	    // decoding of EFPC modus
	    CASE BYTE_TO_INT(#FML_REF.FPCS_Modus) OF
	        0: (* old style *)
	            (* 
	            -------------- Byte 1 --------------- Byte 2 ---------------------- Byte 3/4 ------------------- Byte 5..8 ----
	            |  8  7  6  5  4  |  3  2  1  0  |              | 15 14 13 12 |  11  | 10 9 8 7 6 5 4 3 2 1 0 |               |
	            |    FPCS Modus   |     res      |   Subindex   |      AK     |  SPM |        PNU             |     Value     |
	            ---------------------------------------------------------------------------------------------------------------     
	            AK:  Response Identifier (Antwortkennung)
	            SPM: NOT used
	            PNU: Parameternummer / Parameter-Number 
	            *)
	            // Byte1
	            // zero in this CASE
	            // Byte2  
	            #FML_REF.ActSubindex := #FML_REF.InData.FPC[2];
	            
	            // Byte3/4
	            #BByte2[1] := #FML_REF.InData.FPC[3];
	            #BByte2[2] := #FML_REF.InData.FPC[4];
	            #Resp_Identifier := WORD_TO_INT(SHR(IN := (#_Word AND 2#1111000000000000), N := 12));
	            #FML_REF.ActPNU := #_Word AND 2#0000011111111111;
	            
	            // Byte 5..8 parameter value
	            #BByte4[1] := #FML_REF.InData.FPC[5];
	            #BByte4[2] := #FML_REF.InData.FPC[6];
	            #BByte4[3] := #FML_REF.InData.FPC[7];
	            #BByte4[4] := #FML_REF.InData.FPC[8];
	            #FML_REF.ParamValueRD := #_DINT;
	            
	        1, 2, 3:(* modus: 1 = PNU extended; 2 = KO; 3 = CAN Objects *)
	            (* 
	            -------------- Byte 1 --------------- Byte 2 ------------------- Byte 3/4----------------- Byte 5..8 ----
	            |   7  6  5  4  |  3  2  1  0  |              | 15 14 13 12 11 10 9 8 7 6 5 4 3 2 1 0 |               |
	            |  FPCS Modus   |     AK       |   Subindex   |   PNU extended or KO or CAN Object    |     Value     |
	            -------------------------------------------------------------------------------------------------------       
	            AK:  Response Identifier (Antwortkennung)
	            *)
	            
	            // Byte 1 FPCS
	            #Resp_Identifier := WORD_TO_INT(#FML_REF.InData.FPC[1] AND 2#00001111);
	            
	            // Byte 2 Subindex
	            #FML_REF.ActSubindex := #FML_REF.InData.FPC[2];
	            
	            // Byte 3+4 **PKE/ PNU/ KO/ CAN**
	            #BByte2[1] := #FML_REF.InData.FPC[3];
	            #BByte2[2] := #FML_REF.InData.FPC[4];
	            #FML_REF.ActPNU := #_Word;
	            
	            // Byte 5..8 parameter value
	            #BByte4[1] := #FML_REF.InData.FPC[5];
	            #BByte4[2] := #FML_REF.InData.FPC[6];
	            #BByte4[3] := #FML_REF.InData.FPC[7];
	            #BByte4[4] := #FML_REF.InData.FPC[8];
	            #FML_REF.ParamValueRD := #_DINT;
	            
	        4, 5:(* FPCS_Modus 4=Parameter File; 5=Firmware File *)
	            (*
	            ------ BYTE 1 ------------|-- BYTE 2 -|--BYTE 3..8 ---|
	            | 7  6  5  4 | 3  2  1  0 |           |               |
	            | FPCS Modus |   res      | Packet-ID |  6 BYTE Data  |
	            -------------------------------------------------------        
	              Packet-ID: -------------- BYTE 2 ----------
	                         | 7    6    5  | 4  3  2  1  0 |
	                         | Control Bits |   Sequence-Nr |
	                         -------------------------------- 
	            *)
	            // Byte 1 FPCS
	            #Resp_Identifier := WORD_TO_INT(#FML_REF.InData.FPC[1] AND 2#00001111);
	            #FML_REF.RespID := #Resp_Identifier;
	            
	            //---- Byte 2 Packet-ID ----    
	            #FML_REF.FPCS_Packet.BitSequenceNr := WORD_TO_INT(#FML_REF.InData.FPC[2] AND 2#00011111);
	            #FML_REF.FPCS_Packet.Control := WORD_TO_INT(SHR(IN := (#FML_REF.InData.FPC[2] AND 2#11100000), N := 5));
	            //---- Byte 3..8 Data ----
	            #FML_REF.FPCS_Packet.Data[1] := #FML_REF.InData.FPC[3];
	            #FML_REF.FPCS_Packet.Data[2] := #FML_REF.InData.FPC[4];
	            #FML_REF.FPCS_Packet.Data[3] := #FML_REF.InData.FPC[5];
	            #FML_REF.FPCS_Packet.Data[4] := #FML_REF.InData.FPC[6];
	            #FML_REF.FPCS_Packet.Data[5] := #FML_REF.InData.FPC[7];
	            #FML_REF.FPCS_Packet.Data[6] := #FML_REF.InData.FPC[8];
	            
	            
	        ELSE (* not implemented *)
	            #FPC_MAPPING := FALSE; (* Execution was not correct *)
	            RETURN;
	    END_CASE;
	    
	    CASE #Resp_Identifier OF
	        0, 3:(* No Transmission or Active*)
	            #FML_REF.Done := FALSE;
	            #FML_REF.Err := FALSE;
	            #FML_REF.ActPNU := 0;
	            #FML_REF.ActSubindex := 0;
	            #FML_REF.ParamValueRD := 0;
	            #FML_REF.DatatypeRD := 0;
	            
	            
	        1, 4:(* Word Parameter transmittead*)
	            #FML_REF.Done := TRUE;
	            #FML_REF.Err := FALSE;
	            #FML_REF.ParamValueRD := #_DINT;
	            #FML_REF.DatatypeRD := 2;
	            
	        2, 5: (*DWord Parameter transmitted*)
	            #FML_REF.Done := true;
	            #FML_REF.Err := FALSE;
	            #FML_REF.ParamValueRD := #_DINT;
	            #FML_REF.DatatypeRD := 4;
	            
	        7:(* Transmission Failed*)
	            #FML_REF.Done := TRUE;
	            #FML_REF.Err := TRUE;
	            #FML_REF.DatatypeRD := 0;
	            #FML_REF.ParamValueRD := 0;
	            #FML_REF.ActPNU := 0;
	            
	            
	        11, 12: (*BYTE Parameter transmitted*)
	            #FML_REF.Done := TRUE;
	            #FML_REF.Err := False;
	            #FML_REF.DatatypeRD := 1;
	            #FML_REF.ParamValueRD := #_DINT;
	            
	        ELSE (* not specified*)
	            #FML_REF.Done := false;
	            #FML_REF.Err := TRUE;
	            #FML_REF.ParamValueRD := 0;
	    END_CASE;
	    
	    #FPC_MAPPING := TRUE; (* Execution was correct *)
	    RETURN;
	    
	(* MAP OUTPUTS *)
	ELSE
	    
	    IF #FML_REF.DeviceType = 'SFC_DC' OR #FML_REF.DeviceType = 'MTR_DCI' THEN
	        IF #FML_REF.ReqID = 8 THEN // write
	            IF BYTE_TO_INT(#FML_REF.Subindex) > 0 THEN
	                CASE BYTE_TO_INT(#FML_REF.DatatypeWR) OF
	                    1:
	                        #FML_REF.ReqID := 12;     //Array-Byte
	                    2:
	                        #FML_REF.ReqID := 7;      //Array-Wort
	                    4:
	                        #FML_REF.ReqID := 8;      //Array-Doppelwort
	                    ELSE
	                        #FPC_MAPPING := FALSE; (* wrong data type*)
	                        RETURN;
	                END_CASE;
	            END_IF;
	            (*WRITE SINGLE PARAMETER*)
	            IF #FML_REF.Subindex = 0 THEN
	                CASE BYTE_TO_INT(#FML_REF.DatatypeWR) OF
	                    1:
	                        #FML_REF.ReqID := 11;       // Single-Byte
	                    2:
	                        #FML_REF.ReqID := 2;        // Single-Wort
	                    4:
	                        #FML_REF.ReqID := 3;        // Single-Doppelwort
	                    ELSE
	                        #FPC_MAPPING := FALSE; (* wrong data type*)
	                        RETURN;
	                END_CASE;
	            END_IF;
	            
	        ELSIF #FML_REF.ReqID = 6 THEN
	            (* READ ARRAY PARAMETER *)
	            IF BYTE_TO_INT(#FML_REF.Subindex) > 0 THEN
	                #FML_REF.ReqID := 6;
	            END_IF;
	            (* READ SINGLE PARAMETER *)
	            IF #FML_REF.Subindex = 0 THEN
	                #FML_REF.ReqID := 1;
	            END_IF;
	        ELSE
	            ;// not specified
	        END_IF;
	    END_IF;
	    (* create request identifier *)
	    #Req_Identifier := #FML_REF.ReqID;
	    
	    CASE BYTE_TO_INT(#FML_REF.FPCC_Modus) OF
	        0: (* old style *)
	            (* 
	            -------------- Byte 1 --------------- Byte 2 ---------------------- Byte 3 --------------------- Byte 5..8 ----
	            |  8  7  6  5  4  |  3  2  1  0  |              | 15 14 13 12 |  11  | 10 9 8 7 6 5 4 3 2 1 0 |               |
	            |    FPCS Modus   |     res      |   Subindex   |      AK     |  SPM |        PNU             |     Value     |
	            ---------------------------------------------------------------------------------------------------------------     
	            AK:  Request Identifier (Auftragskennung)
	            SPM: NOT used
	            PNU: Parameternummer / Parameter-Number 
	            *)
	            (* Byte 1 *)
	            #FML_REF.OutData.FPC[1] := SHL(IN := #FML_REF.FPCC_Modus, N := 4);
	            (* Byte 2 Subindex *)
	            #FML_REF.OutData.FPC[2] := #FML_REF.Subindex;
	            (* Byte 3+4 *)
	            #_Word := SHL(IN := INT_TO_WORD(#Req_Identifier), N := 12) OR (#FML_REF.PNU AND 16#07_FF);
	            
	            (* Byte 5..8 *)
	            #_DINT := #FML_REF.ParamValueWR;
	            #FML_REF.OutData.FPC[3] := #BByte2[1]; //Convert PKE to Byte
	            #FML_REF.OutData.FPC[4] := #BByte2[2];
	            
	            (* Set Output DATA OF DRIVE *)
	            #FML_REF.OutData.FPC[5] := #BByte4[1]; //Convert PWE to Byte
	            #FML_REF.OutData.FPC[6] := #BByte4[2];
	            #FML_REF.OutData.FPC[7] := #BByte4[3];
	            #FML_REF.OutData.FPC[8] := #BByte4[4];
	            
	        1, 2, 3:(* modus: 1 = PNU extended; 2 = KO; 3 = CAN Objects *)
	            (* 
	            -------------- Byte 1 --------------- Byte 2 ------------------- Byte 3 ------------------ Byte 5..8 ----
	            |  8  7  6  5  4  |  3  2  1  0  |              | 15 14 13 12 11 10 9 8 7 6 5 4 3 2 1 0 |               |
	            |    FPCS Modus   |     AK       |   Subindex   |   PNU extended or KO or CAN Object    |     Value     |
	            ---------------------------------------------------------------------------------------------------------       
	            AK:  Request Identifier (Auftragskennung)
	            *)
	            (* Byte 1 *)
	            #FML_REF.OutData.FPC[1] := WORD_TO_BYTE(SHL(IN := #FML_REF.FPCC_Modus, N := 4) OR INT_TO_WORD(#Req_Identifier));
	            (* Byte 2 Subindex *)
	            #FML_REF.OutData.FPC[2] := #FML_REF.Subindex;
	            (* Byte 3+4 *)
	            #_Word := #FML_REF.PNU;
	            (* Byte 5..8 *)
	            #_DINT := #FML_REF.ParamValueWR;
	            #FML_REF.OutData.FPC[3] := #BByte2[1]; //Convert PKE to Byte
	            #FML_REF.OutData.FPC[4] := #BByte2[2];
	            
	            (* Set Output DATA OF DRIVE *)
	            #FML_REF.OutData.FPC[5] := #BByte4[1]; //Convert PWE to Byte
	            #FML_REF.OutData.FPC[6] := #BByte4[2];
	            #FML_REF.OutData.FPC[7] := #BByte4[3];
	            #FML_REF.OutData.FPC[8] := #BByte4[4];
	            
	        4, 5:(* FPCC_Modus 4=parameter file; 5=firmware file     
	        |---------- byte 1 --------|-- byte 2 --|-- byte 3..8 ---|
	        | 7  6  5  4  | 3  2  1  0 |            |                |
	        |   FPCC modus |   res      | packet-ID  |  6 byte data  |
	        ---------------------------------------------------------       
	        Packet-ID:  | 7    6    5  | 4  3  2  1  0  |
	                    | control bits |  sequence-nr   |
	                    --------------------------------- *)
	                    //---- byte 1 ----
	                    #FML_REF.OutData.FPC[1] := WORD_TO_BYTE(SHL(IN := #FML_REF.FPCC_Modus, N := 4) OR INT_TO_WORD(#Req_Identifier));
	                    //----byte 2 packet-ID ---- 
	                    #FML_REF.OutData.FPC[2] := (SHL(IN := INT_TO_BYTE(#FML_REF.FPCC_Packet.Control), N := 5) OR (INT_TO_BYTE(#FML_REF.FPCC_Packet.BitSequenceNr) AND 16#1F));
	                    //---- byte 3..8 data ----
	                    #FML_REF.OutData.FPC[3] := #FML_REF.FPCC_Packet.Data[1];         // byte swapping for modbus data 
	                    #FML_REF.OutData.FPC[4] := #FML_REF.FPCC_Packet.Data[2];
	                    #FML_REF.OutData.FPC[5] := #FML_REF.FPCC_Packet.Data[3];
	                    #FML_REF.OutData.FPC[6] := #FML_REF.FPCC_Packet.Data[4];
	                    #FML_REF.OutData.FPC[7] := #FML_REF.FPCC_Packet.Data[5];
	                    #FML_REF.OutData.FPC[8] := #FML_REF.FPCC_Packet.Data[6];
	                    
	                ELSE (* not implemented *)
	                    #FPC_MAPPING := FALSE; (* Execution was not correct *)
	                    RETURN;
	            END_CASE;
	            
	            #FPC_MAPPING := TRUE; (* Execution was correct *)
	        END_IF;
	        
END_FUNCTION

FUNCTION "FHPPPLUS_MAPPING" : DInt
{ S7_Optimized_Access := 'TRUE' }
AUTHOR : FESTO
FAMILY : 'E-DRIVES'
VERSION : 5.1
   VAR_INPUT 
      cfgFHPPplus : DInt;
   END_VAR

   VAR_OUTPUT 
      FHPPplusElementSize : Array[1..9] of DInt;
      FHPPplusSize : DInt;
   END_VAR

   VAR_TEMP 
      i : Int;
      n : Int;
      tmpTeiler : DInt;
      tmpCfgFHPPplus : DInt;
      tmpElementSize : DInt;
      tmpFHPPplusSize : DInt;
   END_VAR

   VAR CONSTANT 
      constTeiler : DInt := 100_000_000;
   END_VAR


BEGIN
	(*############################################################
	   FESTO AG  Co., Esslingen
	   Copyright (c) 2015. All rights reserved.    
	
	   NAME OF FUNCTION BLOCK:         FHPPPLUS_MAPPING
	   VERSION NUMBER:                 V5.1
	   COMPOSER:                       bejk
	   
	       
	   -----------------------------------------------------
	   Date        Name                Activity                                                                              
	   06.08.2015  Benjamin Kilgus     created (V1.0)
	   29.08.2016  Benjamin Klein      version changed (V4.1)
	   05.07.2017  Benjamin Klein      changed to optimized access (V5.1)
	 
	############################################################*)
	
	#tmpTeiler := #constTeiler;
	#tmpCfgFHPPplus := #cfgFHPPplus;
	#tmpFHPPplusSize := 0;
	#n := 1;
	
	// configuration 0 is not legal
	IF #cfgFHPPplus = 0 THEN
	    #FHPPPLUS_MAPPING := DWORD_TO_DINT(16#8000_0001);
	    RETURN;
	END_IF;
	
	FOR #i := 1 TO 9 DO
	    #tmpElementSize := #tmpCfgFHPPplus / #tmpTeiler;
	    IF #tmpElementSize = 1 OR #tmpElementSize = 2 OR #tmpElementSize = 4 THEN
	        #FHPPplusElementSize[#n] := #tmpElementSize * 8; // Byte *8 = Bit
	        #tmpFHPPplusSize := #tmpFHPPplusSize + #FHPPplusElementSize[#n];
	        #tmpCfgFHPPplus := #tmpCfgFHPPplus - (#tmpElementSize * #tmpTeiler);
	        #n := #n + 1;
	    ELSIF #tmpElementSize = 0 AND #n = 1 THEN // digit empty
	        #FHPPplusElementSize[10 - #i] := 0;
	    ELSE
	        #FHPPPLUS_MAPPING := DWORD_TO_DINT(16#8000_0001); // wrong configuration
	        RETURN;
	    END_IF;
	    #tmpTeiler := #tmpTeiler / 10;
	END_FOR;
	
	IF #tmpFHPPplusSize = 64 OR #tmpFHPPplusSize = 128 OR #tmpFHPPplusSize = 192 THEN
	    ;// o.k.
	    
	ELSE // wrong size
	    #FHPPPLUS_MAPPING := DWORD_TO_DINT(16#8000_0001); // function is called without legal FHPP+ configuration
	    RETURN;
	END_IF;
	
	#FHPPplusSize := #tmpFHPPplusSize;
	#FHPPPLUS_MAPPING := 0; // o.k.
	
END_FUNCTION

FUNCTION_BLOCK "FHPP_CTRL"
{ S7_Optimized_Access := 'TRUE' }
AUTHOR : FESTO
FAMILY : 'E-DRIVE'
VERSION : 5.1
   VAR_INPUT 
      EnableDrive : Bool;
      Stop : Bool;
      Halt : Bool;
      Brake : Bool;
      ResetFault : Bool;
      HMIAccessLocked : Bool;
      OPM : Int;
      StartTask : Bool;
      StartHoming : Bool;
      JogPos : Bool;
      JogNeg : Bool;
      TeachActValue : Bool;
      ClearRemPos : Bool;
      Relative : Bool;
      DeactivateStrokeLimit : Bool;
      ExecuteFunction : Bool;
      RecordNo : Int;
      SetFunctionNumber : Int;
      SetFunctionGroup : Int;
      SetValueVelocity : DInt;
      SetValuePosition : DInt;
      SetValueForceRamp : DInt;
      SetValueForce : DInt;
      SetValueRotRamp : DInt;
      SetValueRotSpeed : DInt;
   END_VAR

   VAR_OUTPUT 
      DriveEnabled : Bool;
      Ready : Bool;
      Warning : Bool;
      Fault : Bool;
      SupplyVoltPresent : Bool;
      ControlFCT_HMI : Bool;
      StateOPM : Int;
      HaltNotActive : Bool;
      AckStart : Bool;
      MC : Bool;
      AckTeach : Bool;
      DriveMoving : Bool;
      DragError : Bool;
      StandStillControl : Bool;
      HomingValid : Bool;
      ActualRecordNo : Int;
      RC1 : Bool;
      RCC : Bool;
      VelocityLimitReached : Bool;
      StrokeLimitReached : Bool;
      FunctionIsActive : Bool;
      ActualFunctionNumber : Int;
      ActualFunctionGroup : Int;
      ActualPosition : DInt;
      ActualVelocity : DInt;
      ActualForce : DInt;
      ActualRotRamp : DInt;
      ActualRotSpeed : DInt;
   END_VAR

   VAR_IN_OUT 
      FML_REF : "DT_FML_REF";
   END_VAR

   VAR 
      Converted_BYTE5_8_IN : DInt;
      Converted_BYTE5_8_OUT : DInt;
      OperationModeB1 : Bool;
      OperationModeB2 : Bool;
      ControlModeB1 : Bool;
      ControlModeB2 : Bool;
      ContinuousMode : Bool;
      StateOperationModeB1 : Bool;
      StateOperationModeB2 : Bool;
      StateControlModeB1 : Bool;
      StateControlModeB2 : Bool;
      StateContinuousMode : Bool;
   END_VAR

   VAR_TEMP 
      tmpDevice : String[16];
   END_VAR


BEGIN
	(*############################################################
	   FESTO AG  Co., Esslingen
	   Copyright (c) 2015. All rights reserved.    
	
	   NAME OF FUNCTION BLOCK:         FHPP_CTRL
	   VERSION NUMBER:                 V5.1
	   COMPOSER:                       bejk
	   
	         
	   -----------------------------------------------------
	   Date        Name                Activity                                                                              
	   15.04.2015  Benjamin Kilgus     converted from Step7 V5.5 (V3.0)
	   25.08.2015  Benjamin Kilgus     ActualVelocity, cast changed to BYTE_TO_SINT 
	                                   case 5 for SetValue's adjusted to FW specific differents (V3.1)
	   16.11.2015  Benjamin Kilgus     Änderungen für kompatibilität S7300/S7400 (V3.2)   
	   13.04.2016  Benjamin Klein      Änderungen für FUNC Bit hinzugefügt
	   01.08.2016  Benjamin Klein      SetValueForce wird auf 120% begrenzt, da die Rückmeldung nur 1 Byte Wertebereich hat.
	   12.08.2016  Benjamin Klein      Datentyp ActualVelocity,ActualForce und ActualRotRamp auf INT geändert. 
	   29.08.2016  Benjamin Klein      version changed (V4.1)
	   21.09.2016  Benjamin Klein      bugfix Actual Force, limit in SetForce deactivated, SetFunctionNumber bugfix (V4.2)
	   16.03.2016  Benjamin Klein      optimized function block with Slice access instead of AT (V5.1)
	############################################################*)
	
	(*-----------------------------------------------------------
	    Initial Block Routine
	------------------------------------------------------------*)
	#tmpDevice := #FML_REF.DeviceType;
	
	(* Byte_3 *)
	#StrokeLimitReached := FALSE;
	#VelocityLimitReached := FALSE;
	#StateContinuousMode := FALSE;
	#StateControlModeB2 := FALSE;
	#StateControlModeB1 := FALSE;
	#ActualRecordNo := 0;
	
	(* Byte_4 *)
	#RC1 := FALSE;
	#RCC := FALSE;
	#VelocityLimitReached := FALSE;
	#StrokeLimitReached := FALSE;
	
	#ActualVelocity := 0;
	#ActualForce := 0;
	#ActualRotRamp := 0;
	
	(* Byte5-8 *)
	#ActualPosition := 0;
	#ActualRotSpeed := 0;
	
	(*-----------------------------------------------------------
	    Asignment of the Input Data (Stateword)
	------------------------------------------------------------*)
	#Converted_BYTE5_8_IN.%B3 := #FML_REF.InData.FHPP[5];
	#Converted_BYTE5_8_IN.%B2 := #FML_REF.InData.FHPP[6];
	#Converted_BYTE5_8_IN.%B1 := #FML_REF.InData.FHPP[7];
	#Converted_BYTE5_8_IN.%B0 := #FML_REF.InData.FHPP[8];
	
	
	(* Byte1 SCON *)
	
	#StateOperationModeB2 := #FML_REF.InData.FHPP[1].%X7;
	#StateOperationModeB1 := #FML_REF.InData.FHPP[1].%X6;
	#ControlFCT_HMI := #FML_REF.InData.FHPP[1].%X5;
	#SupplyVoltPresent := #FML_REF.InData.FHPP[1].%X4;
	#Fault := #FML_REF.InData.FHPP[1].%X3;
	#Warning := #FML_REF.InData.FHPP[1].%X2;
	#Ready := #FML_REF.InData.FHPP[1].%X1;
	#DriveEnabled := #FML_REF.InData.FHPP[1].%X0;
	
	(* Byte2 SPOS *)
	
	#HomingValid := #FML_REF.InData.FHPP[2].%X7;
	#StandStillControl := #FML_REF.InData.FHPP[2].%X6;
	#DragError := #FML_REF.InData.FHPP[2].%X5;
	#DriveMoving := #FML_REF.InData.FHPP[2].%X4;
	#AckTeach := #FML_REF.InData.FHPP[2].%X3;
	#MC := #FML_REF.InData.FHPP[2].%X2;
	#AckStart := #FML_REF.InData.FHPP[2].%X1;
	#HaltNotActive := #FML_REF.InData.FHPP[2].%X0;
	
	(* Byte_3 *)
	IF #StateOperationModeB1 THEN        // ===== directmode active =====
	(* SDIR *)
	    
	    IF #FML_REF.InData.FHPP[3].%X7 AND #tmpDevice = 'CMMP_AS' THEN
	        
	        IF #FML_REF.InData.FHPP[3].%X3 AND #FML_REF.InData.FHPP[3].%X4 THEN
	            #ActualFunctionNumber := 3;
	        ELSIF NOT #FML_REF.InData.FHPP[3].%X3 AND #FML_REF.InData.FHPP[3].%X4 THEN
	            #ActualFunctionNumber := 2;
	        ELSIF #FML_REF.InData.FHPP[3].%X3 AND NOT #FML_REF.InData.FHPP[3].%X4 THEN
	            #ActualFunctionNumber := 1;
	        ELSE
	            #ActualFunctionNumber := 0;
	        END_IF;
	        
	        IF #FML_REF.InData.FHPP[3].%X5 AND #FML_REF.InData.FHPP[3].%X6 THEN
	            #ActualFunctionGroup := 3;
	        ELSIF NOT #FML_REF.InData.FHPP[3].%X5 AND #FML_REF.InData.FHPP[3].%X6 THEN
	            #ActualFunctionGroup := 2;
	        ELSIF #FML_REF.InData.FHPP[3].%X5 AND NOT #FML_REF.InData.FHPP[3].%X6 THEN
	            #ActualFunctionGroup := 1;
	        ELSE
	            #ActualFunctionGroup := 0;
	        END_IF;
	        
	        #FunctionIsActive := TRUE;
	        #StateControlModeB2 := #FML_REF.InData.FHPP[3].%X2;
	        #StateControlModeB1 := #FML_REF.InData.FHPP[3].%X1;
	        ;
	    ELSE
	        #StrokeLimitReached := #FML_REF.InData.FHPP[3].%X5;
	        #VelocityLimitReached := #FML_REF.InData.FHPP[3].%X4;
	        #StateContinuousMode := #FML_REF.InData.FHPP[3].%X3;
	        #StateControlModeB2 := #FML_REF.InData.FHPP[3].%X2;
	        #StateControlModeB1 := #FML_REF.InData.FHPP[3].%X1;
	        
	        #FunctionIsActive := FALSE;
	        #ActualFunctionNumber := 0;
	        #ActualFunctionGroup := 0;
	    END_IF;
	ELSE                                // ===== recordmode active =====
	(* RecordNo *)
	    #ActualRecordNo := BYTE_TO_INT(#FML_REF.InData.FHPP[3]);
	    
	    #FunctionIsActive := FALSE;
	    #ActualFunctionNumber := 0;
	    #ActualFunctionGroup := 0;
	    ;
	END_IF;
	
	(* Coding of the Operation Mode State *)
	#StateOPM := 0;
	#StateOPM.%X0 := #StateOperationModeB1;
	#StateOPM.%X1 := #StateOperationModeB2;
	#StateOPM.%X2 := #StateControlModeB1;
	#StateOPM.%X3 := #StateControlModeB2;
	#StateOPM.%X4 := #StateContinuousMode;
	
	
	(* Byte_4/ Byte5-8*)
	CASE #StateOPM OF
	    0:// (0)  Recordmode
	        (* RSB record state *)
	        
	        #RC1 := #FML_REF.InData.FHPP[4].%X0;
	        #RCC := #FML_REF.InData.FHPP[4].%X1;
	        #VelocityLimitReached := #FML_REF.InData.FHPP[4].%X4;
	        #StrokeLimitReached := #FML_REF.InData.FHPP[4].%X5;
	        #ActualPosition := #Converted_BYTE5_8_IN;
	        
	    1:
	        // (1)  Directmode Position Control
	        #ActualVelocity := SINT_TO_DINT(#FML_REF.InData.FHPP[4]);
	        #ActualPosition := #Converted_BYTE5_8_IN;
	        
	    5:// Directmode Force Control 
	        
	        #ActualForce := SINT_TO_DINT(#FML_REF.InData.FHPP[4]);
	        #ActualPosition := #Converted_BYTE5_8_IN;
	        
	    9:// Directmode Rotation-Speed-Control
	        #ActualRotRamp := SINT_TO_DINT(#FML_REF.InData.FHPP[4]);
	        #ActualRotSpeed := #Converted_BYTE5_8_IN;
	    ELSE
	        ;
	END_CASE;
	
	(*-----------------------------------------------------------
	    Asignment of the Output Data (Controlword)
	------------------------------------------------------------*)
	(* Decoding of the Operationmode *)
	//#_Word := INT_TO_WORD(#OPM);
	#OperationModeB1 := #OPM.%X0;
	#OperationModeB2 := #OPM.%X1;
	#ControlModeB1 := #OPM.%X2;
	#ControlModeB2 := #OPM.%X3;
	#ContinuousMode := #OPM.%X4;
	
	
	(* CCON Byte_1 *)
	#FML_REF.OutData.FHPP[1].%X7 := #OperationModeB2;
	#FML_REF.OutData.FHPP[1].%X6 := #OperationModeB1; // selection of Operation Mode
	#FML_REF.OutData.FHPP[1].%X5 := #HMIAccessLocked; // get control sovereignty
	#FML_REF.OutData.FHPP[1].%X4 := false;
	#FML_REF.OutData.FHPP[1].%X3 := #ResetFault;
	#FML_REF.OutData.FHPP[1].%X2 := #Brake;
	#FML_REF.OutData.FHPP[1].%X1 := #Stop;
	#FML_REF.OutData.FHPP[1].%X0 := #EnableDrive;
	
	
	(* CPOS Byte_2 *)
	#FML_REF.OutData.FHPP[2].%X7 := FALSE;
	#FML_REF.OutData.FHPP[2].%X6 := #ClearRemPos;
	#FML_REF.OutData.FHPP[2].%X5 := #TeachActValue;
	#FML_REF.OutData.FHPP[2].%X4 := #JogNeg;
	#FML_REF.OutData.FHPP[2].%X3 := #JogPos;
	#FML_REF.OutData.FHPP[2].%X2 := #StartHoming;
	#FML_REF.OutData.FHPP[2].%X1 := #StartTask;
	#FML_REF.OutData.FHPP[2].%X0 := #Halt;
	
	(* Byte_3 *)
	IF #OperationModeB1 THEN     // ===== directmode =====
	(* CDIR *)
	    IF #ExecuteFunction AND #tmpDevice = 'CMMP_AS' THEN
	        #FML_REF.OutData.FHPP[3].%X7 := TRUE;                                          // CDIR_B7:FUNC
	        #FML_REF.OutData.FHPP[3].%X6 := false;                                     // Func Group actually not used
	        #FML_REF.OutData.FHPP[3].%X5 := false;                                     // Func Group actually not used
	        IF #SetFunctionNumber = 3 THEN
	            #FML_REF.OutData.FHPP[3].%X4 := TRUE;
	            #FML_REF.OutData.FHPP[3].%X3 := TRUE;
	        ELSIF #SetFunctionNumber = 2 THEN
	            #FML_REF.OutData.FHPP[3].%X4 := TRUE;
	            #FML_REF.OutData.FHPP[3].%X3 := FALSE;
	        ELSIF #SetFunctionNumber = 1 THEN
	            #FML_REF.OutData.FHPP[3].%X4 := FALSE;
	            #FML_REF.OutData.FHPP[3].%X3 := TRUE;
	        ELSE
	            #FML_REF.OutData.FHPP[3].%X4 := FALSE;
	            #FML_REF.OutData.FHPP[3].%X3 := false;
	        END_IF;
	        #FML_REF.OutData.FHPP[3].%X2 := #ControlModeB2;
	        #FML_REF.OutData.FHPP[3].%X1 := #ControlModeB1;
	        #FML_REF.OutData.FHPP[3].%X0 := #Relative;
	        
	    ELSE
	        #FML_REF.OutData.FHPP[3].%X7 := FALSE;
	        #FML_REF.OutData.FHPP[3].%X6 := FALSE;
	        #FML_REF.OutData.FHPP[3].%X5 := #DeactivateStrokeLimit;
	        #FML_REF.OutData.FHPP[3].%X4 := FALSE;
	        #FML_REF.OutData.FHPP[3].%X3 := FALSE;
	        #FML_REF.OutData.FHPP[3].%X2 := #ControlModeB2;
	        #FML_REF.OutData.FHPP[3].%X1 := #ControlModeB1;
	        #FML_REF.OutData.FHPP[3].%X0 := #Relative;
	    END_IF;
	ELSE                        // ===== recordmode =====
	(* RecordNo *)
	    #FML_REF.OutData.FHPP[3] := INT_TO_BYTE(#RecordNo);
	END_IF;
	
	(* Byte4/ Byte5-8 *)
	CASE #OPM OF
	    0:// (0)  Recordmode
	        #FML_REF.OutData.FHPP[4] := 0;
	        #Converted_BYTE5_8_OUT := 0;
	        
	    1:
	        // (1)  Directmode Position Control
	        #FML_REF.OutData.FHPP[4] := DINT_TO_BYTE(MIN(IN1 := #SetValueVelocity, IN2 := 100));                   // byte 4 (permissible range of value is 0 to 100)
	        #Converted_BYTE5_8_OUT := #SetValuePosition;
	        
	    5:// Directmode Forcecontrol
	        (* CMMP-AS *)
	        IF (#tmpDevice = 'CMMP_AS') THEN
	            #FML_REF.OutData.FHPP[4] := DINT_TO_BYTE(MIN(IN1 := #SetValueForceRamp, IN2 := 100));          // byte 4 (permissible range of value is 0 to 100);
	            (* CMMO-ST AND EMCA-EC *)
	        ELSIF (#tmpDevice = 'CMMO_ST') OR (#tmpDevice = 'EMCA_EC') THEN
	            #FML_REF.OutData.FHPP[4] := DINT_TO_BYTE(MIN(IN1 := #SetValueVelocity, IN2 := 100));
	            (*other*)
	        ELSE
	            #FML_REF.OutData.FHPP[4] := 0;
	        END_IF;
	        
	        #Converted_BYTE5_8_OUT := #SetValueForce;
	        
	        
	    9:// Directmode Rotation-Speed-Control      
	        #FML_REF.OutData.FHPP[4] := DINT_TO_BYTE(MIN(IN1 := #SetValueRotRamp, IN2 := 100));                     // byte 4 (permissible range of value is 0 to 100)
	        #Converted_BYTE5_8_OUT := #SetValueRotSpeed;
	        
	    ELSE // illegal OPM              
	        #FML_REF.OutData.FHPP[4] := 0;
	        #Converted_BYTE5_8_OUT := 0;
	END_CASE;
	
	(* Set Output DATA OF DRIVE *)
	#FML_REF.OutData.FHPP[5] := #Converted_BYTE5_8_OUT.%B3;
	#FML_REF.OutData.FHPP[6] := #Converted_BYTE5_8_OUT.%B2;
	#FML_REF.OutData.FHPP[7] := #Converted_BYTE5_8_OUT.%B1;
	#FML_REF.OutData.FHPP[8] := #Converted_BYTE5_8_OUT.%B0;
	
	
	
	
	
	
	
	
	
	
	
	
	
END_FUNCTION_BLOCK

FUNCTION_BLOCK "FHPP_DPWR_DAT"
{ S7_Optimized_Access := 'TRUE' }
AUTHOR : FESTO
FAMILY : 'E-DRIVE'
VERSION : 5.1
   VAR_INPUT 
      HW_IO_FHPP : HW_IO;
      HW_IO_FPC : HW_IO;
   END_VAR
   VAR_INPUT DB_SPECIFIC
      HW_IO_FHPPplus : HW_IO;
      cfgFHPPplusOut : DInt;
   END_VAR

   VAR_OUTPUT 
      Error : Bool;
      Status : "DT_FML_STATUS";
   END_VAR

   VAR_IN_OUT 
      FML_REF : "DT_FML_REF";
   END_VAR

   VAR 
      EnableFHPPplusOutOld : DInt;
      FHPPplusSize { ExternalAccessible := 'False'; ExternalVisible := 'False'; ExternalWritable := 'False'} : DInt;
      FHPPplusElementSize { ExternalAccessible := 'False'; ExternalVisible := 'False'; ExternalWritable := 'False'} : Array[1..9] of DInt;
   END_VAR

   VAR_TEMP 
      tmp_bRetVal : Bool;
      iByteCount : Int;
      i : Int;
      FHPPplus8 : Array[1..8] of Byte;
      FHPPplus16 : Array[1..16] of Byte;
      FHPPplus24 : Array[1..24] of Byte;
      WORD_BYTE : Word;
      DWORD_BYTE : DInt;
      tmpStatus : "DT_FML_STATUS";
      tmp_FML_REF : "DT_FML_REF";
   END_VAR


BEGIN
	(*############################################################
	    FESTO AG  Co., Esslingen
	    Copyright (c) 2015. All rights reserved.    
	
	    NAME OF FUNCTION BLOCK:         FHPP_DPWR_DAT
	    VERSION NUMBER:                 V5.1
	    COMPOSER:                       bejk
	    
	    -----------------------------------------------------
	   Date        Name                Activity                                                                              
	   06.08.2015  Benjamin Kilgus     created (V1.0)
	   15.09.2015  Benjamin Kilgus     errorhandling changed (V1.1)
	   29.08.2016  Benjamin Klein      version changed (V4.1)
	   22.09.2016  Benjamin Klein      bugfix: FHPP+ copy 16Byte, tmpStatus.Err initialization  (V4.2)
	   02.11.2016  Benjamin Klein      adapted to TIAV14 (V5.0)  
	   05.07.2017  Benjamin Klein      optimized function block with Slice access instead of AT (V5.1)
	   18.10.2017  Benjamin Klein      "tmpStatus" at beginning deleted, labels deleted
	############################################################*)
	
	// function block (FB) is busy
	#tmpStatus.Err := FALSE;
	#tmpStatus.Cat := 1;
	#tmpStatus.ID := 16#0000_0002; // FB busy 
	
	
	// ### FHPP Standard ##########################################################
	#tmpStatus.Err := false;
	#tmpStatus.ID := INT_TO_WORD(DPWR_DAT(LADDR := #HW_IO_FHPP, RECORD := #FML_REF.OutData.FHPP));
	
	// #Error WHILE reading?
	IF #tmpStatus.ID <> 0 THEN
	    #tmpStatus.Err := TRUE;
	    #tmpStatus.Cat := 4; // SIEMENS
	END_IF;
	
	// ### FHPP FPC ###############################################################
	IF #HW_IO_FPC <> 0 AND #tmpStatus.Err = FALSE THEN
	    
	    // mapping of FPC data 
	    #tmp_FML_REF := #FML_REF;
	    #tmp_bRetVal := NOT "FPC_MAPPING"(Mode := TRUE, FML_REF := #tmp_FML_REF);
	    
	    IF #tmp_bRetVal THEN
	        #tmpStatus.Cat := 3; // FPC
	        #tmpStatus.ID := 18;
	    END_IF;
	    #FML_REF := #tmp_FML_REF;
	    
	    #tmpStatus.ID := INT_TO_WORD(DPWR_DAT(LADDR := #HW_IO_FPC, RECORD := #FML_REF.OutData.FPC));
	    // #Error WHILE reading?
	    IF #tmpStatus.ID <> 0 THEN
	        #tmpStatus.Err := TRUE;
	        #tmpStatus.Cat := 4; // SIEMENS
	    END_IF;
	    
	END_IF;
	
	// ### FHPP PLUS ##########################################################
	IF #HW_IO_FHPPplus <> 0 AND #tmpStatus.Err = FALSE  THEN
	    
	    IF #cfgFHPPplusOut <> #EnableFHPPplusOutOld THEN
	        #tmpStatus.ID := "FHPPPLUS_MAPPING"(cfgFHPPplus := #cfgFHPPplusOut, FHPPplusElementSize => #FHPPplusElementSize, FHPPplusSize => #FHPPplusSize);
	        #EnableFHPPplusOutOld := #cfgFHPPplusOut;
	    END_IF;
	    
	    // FHPP+ Berechnung fehlerhaft beendet
	    IF #tmpStatus.ID <> 0 THEN
	        #tmpStatus.Err := TRUE;
	        #tmpStatus.Cat := 1; // functionblock
	    END_IF;
	    
	    // copy data from FML_REF
	    #iByteCount := 1;
	    FOR #i := 1 TO 9 DO
	        CASE #FHPPplusElementSize[#i] OF
	            0:(* Element is empty *)
	                ;// do nothing
	            8:(* Element is a BYTE *)
	                #FHPPplus24[#iByteCount] := DINT_TO_BYTE(#FML_REF.OutData.FHPPplus[#i]);
	                #iByteCount := #iByteCount + 1;
	            16:(* Element is a WORD *)
	                #WORD_BYTE := DINT_TO_WORD(#FML_REF.OutData.FHPPplus[#i]);
	                #FHPPplus24[#iByteCount] := #WORD_BYTE.%B1;
	                #FHPPplus24[#iByteCount + 1] := #WORD_BYTE.%B0;
	                #iByteCount := #iByteCount + 2;
	            32:(* Element is a DWORD *)
	                #DWORD_BYTE := #FML_REF.OutData.FHPPplus[#i];
	                #FHPPplus24[#iByteCount] := #DWORD_BYTE.%B3;
	                #FHPPplus24[#iByteCount + 1] := #DWORD_BYTE.%B2;
	                #FHPPplus24[#iByteCount + 2] := #DWORD_BYTE.%B1;
	                #FHPPplus24[#iByteCount + 3] := #DWORD_BYTE.%B0;
	                #iByteCount := #iByteCount + 4;
	            ELSE
	                #tmpStatus.Err := TRUE;
	                #tmpStatus.Cat := 1;
	                #tmpStatus.ID := DWORD_TO_DINT(16#8000_0001); // //no legal FHPP+ configuration
	        END_CASE;
	    END_FOR;
	    
	    CASE #FHPPplusSize OF
	        0:(* 0 Byte FHPP+ *)
	            (* NO FHPP+ Data configured *)
	            #tmpStatus.Err := TRUE;
	            #tmpStatus.Cat := 1; // functionblock           
	            #tmpStatus.ID := DWORD_TO_DINT(16#8000_0001); // function is called without legal FHPP+ configuration
	            
	        64: // 8 Byte FHPP+ (64bit)
	            // copy data to FML_REF
	            FOR #i := 1 TO 8 DO
	                #FHPPplus8[#i] := #FHPPplus24[#i];
	            END_FOR;
	            
	            #tmpStatus.ID := INT_TO_WORD(DPWR_DAT(LADDR := #HW_IO_FHPPplus, RECORD := #FHPPplus8));
	            IF #tmpStatus.ID <> 0 THEN
	                #tmpStatus.Err := TRUE;
	                #tmpStatus.Cat := 4; // SIEMENS
	            END_IF;
	        128:// 16 Byte FHPP+ (128bit)
	            // copy data to FML_REF
	            FOR #i := 1 TO 16 DO
	                #FHPPplus16[#i] := #FHPPplus24[#i];
	            END_FOR;
	            
	            #tmpStatus.ID := INT_TO_WORD(DPWR_DAT(LADDR := #HW_IO_FHPPplus, RECORD := #FHPPplus16));
	            IF #tmpStatus.ID <> 0 THEN
	                #tmpStatus.Err := TRUE;
	                #tmpStatus.Cat := 4; // SIEMENS
	            END_IF;
	            
	        192: // 24 Byte FHPP+ (192bit)
	            #tmpStatus.ID := INT_TO_WORD(DPWR_DAT(LADDR := #HW_IO_FHPPplus, RECORD := #FHPPplus24));
	            IF #tmpStatus.ID <> 0 THEN
	                #tmpStatus.Err := TRUE;
	                #tmpStatus.Cat := 4; // SIEMENS
	            END_IF;
	        ELSE
	            #tmpStatus.Err := TRUE;
	            #tmpStatus.Cat := 1;
	            #tmpStatus.ID := DWORD_TO_DINT(16#8000_0001); // function is called without legal FHPP+ configuration
	    END_CASE;
	END_IF;
	
	// ### EXIT ROUTINE ############################################################
	IF NOT #tmpStatus.Err THEN
	    ENO := TRUE;      // Set ENO-Bit to true
	    #Status := #tmpStatus;
	    #Error := #tmpStatus.Err;
	ELSE
	    ENO := FALSE;     // Set ENO-Bit to false
	    #Status := #tmpStatus;
	    #Error := #tmpStatus.Err;
	END_IF;
END_FUNCTION_BLOCK

FUNCTION_BLOCK "CMMS_Z2_Movement"   // FB16, LAD
{ S7_Optimized_Access := 'TRUE' }
VERSION : 0.1
   VAR
      FML_REF : "DT_FML_REF";
   END_VAR
   // FML_REF.DeviceType := 'CMMS';
BEGIN

REGION Network 1
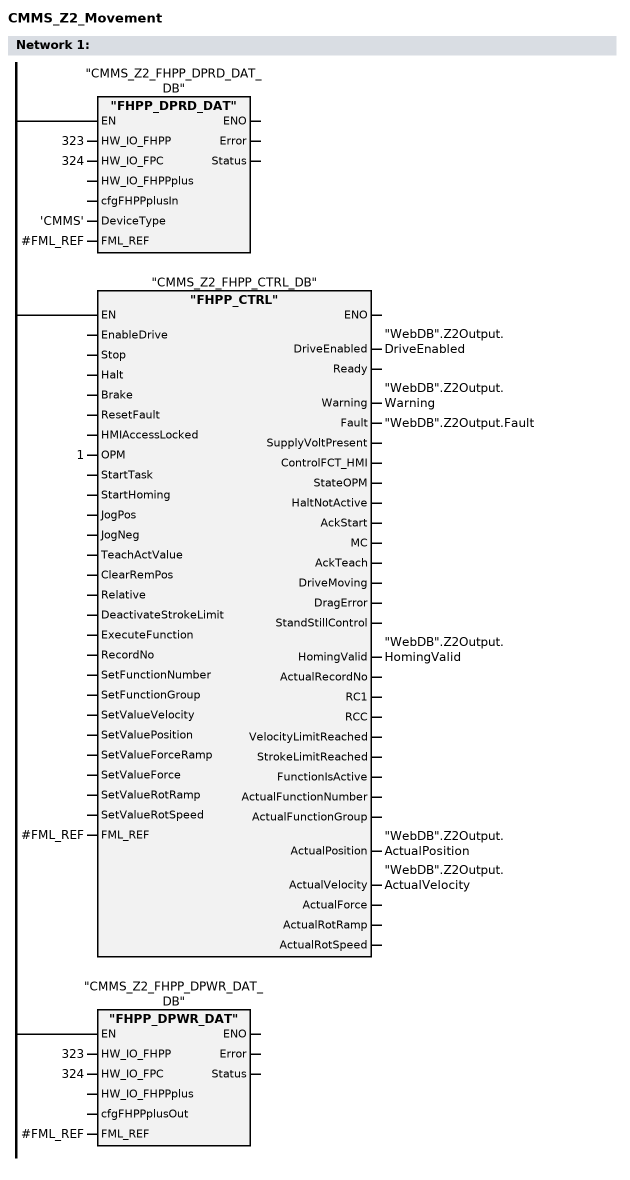
   RUNG wire#powerrail
      "CMMS_Z2_FHPP_DPRD_DAT_DB"(HW_IO_FHPP := 323, HW_IO_FPC := 324, HW_IO_FHPPplus :=, cfgFHPPplusIn :=, DeviceType := 'CMMS', FML_REF := #FML_REF, Error =>, Status =>)
   END_RUNG
   RUNG wire#powerrail
      "CMMS_Z2_FHPP_CTRL_DB"(EnableDrive :=, Stop :=, Halt :=, Brake :=, ResetFault :=, HMIAccessLocked :=, OPM := 1, StartTask :=, StartHoming :=, JogPos :=, JogNeg :=, TeachActValue :=, ClearRemPos :=, Relative :=, DeactivateStrokeLimit :=, ExecuteFunction :=, RecordNo :=, SetFunctionNumber :=, SetFunctionGroup :=, SetValueVelocity :=, SetValuePosition :=, SetValueForceRamp :=, SetValueForce :=, SetValueRotRamp :=, SetValueRotSpeed :=, FML_REF := #FML_REF, DriveEnabled => "WebDB".Z2Output.DriveEnabled, Ready =>, Warning => "WebDB".Z2Output.Warning, Fault => "WebDB".Z2Output.Fault, SupplyVoltPresent =>, ControlFCT_HMI =>, StateOPM =>, HaltNotActive =>, AckStart =>, MC =>, AckTeach =>, DriveMoving =>, DragError =>, StandStillControl =>, HomingValid => "WebDB".Z2Output.HomingValid, ActualRecordNo =>, RC1 =>, RCC =>, VelocityLimitReached =>, StrokeLimitReached =>, FunctionIsActive =>, ActualFunctionNumber =>, ActualFunctionGroup =>, ActualPosition => "WebDB".Z2Output.ActualPosition, ActualVelocity => "WebDB".Z2Output.ActualVelocity, ActualForce =>, ActualRotRamp =>, ActualRotSpeed =>)
   END_RUNG
   RUNG wire#powerrail
      "CMMS_Z2_FHPP_DPWR_DAT_DB"(HW_IO_FHPP := 323, HW_IO_FPC := 324, HW_IO_FHPPplus :=, cfgFHPPplusOut :=, FML_REF := #FML_REF, Error =>, Status =>)
   END_RUNG
   // the same network as SCL:
   "CMMS_Z2_FHPP_DPRD_DAT_DB"(HW_IO_FHPP := 323, HW_IO_FPC := 324, DeviceType := 'CMMS', FML_REF := #FML_REF);   // "FHPP_DPRD_DAT"
   "CMMS_Z2_FHPP_CTRL_DB"(OPM := 1,   // "FHPP_CTRL"
                          FML_REF := #FML_REF,
                          DriveEnabled => "WebDB".Z2Output.DriveEnabled,
                          Warning => "WebDB".Z2Output.Warning,
                          Fault => "WebDB".Z2Output.Fault,
                          HomingValid => "WebDB".Z2Output.HomingValid,
                          ActualPosition => "WebDB".Z2Output.ActualPosition,
                          ActualVelocity => "WebDB".Z2Output.ActualVelocity);
   "CMMS_Z2_FHPP_DPWR_DAT_DB"(HW_IO_FHPP := 323, HW_IO_FPC := 324, FML_REF := #FML_REF);   // "FHPP_DPWR_DAT"
END_REGION
END_FUNCTION_BLOCK

FUNCTION_BLOCK "RollerV3"   // FB2, LAD
TITLE = Description:
{ S7_Optimized_Access := 'TRUE' }
VERSION : 0.1
// How to operate and control the roller:
// Roller is controled by inputs in WebDB: Mode, SetSpeed, Direction, OffsetSpeed. To start the roller use Start_Roller and to stop use Stop_Roller.
// 
// Mode descriptions:
// 0 - Controlling the roller by just turning it ON/OFF
// 1 - Basic speed control of the roller with 0-100%
// 2 - Direct speed control based on Y axis velocity. Not useful for printing, but might help in the development process to observe roller system inertia.
// 3 - Setting relative surface velocity (powder to roller). There is no control loop. Could be used for testing the feature before evaluating.
// 
// E-STOP - always check!
   VAR_INPUT
      "E-STOP" : Bool;
      SystemON : Bool;
      Mode : Int;   // 0 - ON/OFF; 1 - Set Max Speed; 2 - Automatic Yvel=Rvel; 3 - Automatic vel dif
      SetSpeed : Real;   // %
      DirectionLeftRight : Bool;
      Offsetspeed : DInt;
      YAxisVelocity : DInt;
      Roller_HW_address : HW_HSC;
      DoorSensors : Bool;
   END_VAR
   VAR_OUTPUT
      WebDBRollerOutput : Bool;
      RollerDirection : Bool;   // 1 - Clockwise; 0 - Counterclockwise
      RollerLinearVelocity : DInt;   // Microns Per Sec
      RollerRPM : Real;
      RollerRPM_Measured : Real;
   END_VAR
   VAR_IN_OUT
      WebDBStart : Bool;
      WebDBStop : Bool;
   END_VAR
   VAR
      RollerSetReset : Bool;
      RollerFullPower : Bool;
      RollerHalfPower : Bool;
      RollerActive : Bool;
      RollerSpeedInputGeneral : Real;   // %
      RollerSpeedInputPID : Real;
      RollerManualValue : Int;
      Direction_Plus : Bool;   // Clockwise
      Direction_Minus : Bool;   // Counterclockwise
      PulseSignalMeasurement : DWord;
      MaintenanceM3DirDis : Bool := true;
      MaintenanceSkipPID : Bool := true;
      MaintenanceAutomaticDifVel : Bool;   // Change automatic mode from Yvel=Rvel to Difference
      MaintenanceRollerON : Bool;
      RollerDirectionInt_last : Int;
      Roller_RPM_Send_last : Real;
      RollerSetReset_M : Bool;
      RollerSetReset_M2 : Bool;
      hscData : HSC_Period;
   END_VAR
   VAR_TEMP
      DirectionMinusInternal : Bool;
      OffsetSpeedInternal : DInt;
      YAxisVelocityInternal : DInt;
      Roller_Speed_ConvRPM : Real;
      Roller_Speed_ConvPercInput : Real;
      Roller_Speed_ConvDEGSEC : Real;
      Roller_PWM_NormOutput : Real;
      Roller_ConvLinearPerDeg : DInt;
      Roller_Conv_M1_Norm : Real;
      Roller_Conv_M1_Scale : Real;
      Roller_Conv_M2_YvelocityconvRPS : Real;
      Roller_Conv_M2_YvelocityconvRPM : Real;
      Roller_Conv_M3_LinVel : DInt;
      Roller_Conv_M3_Rps : Real;
      Roller_Conv_M3_Rpm : Real;
      Roller_Send_Conv : Real;
      Roller_RPM_Send : Real;
      Roller_RPM_SendRev : Real;
      Roller_Circumference : DInt;   // [microns]
      Roller_Direction_Internal : Bool;
      RollerMinRPMRev : Real;
      RollerDirectionInt : Int;
      ex_vel : Bool;
      RollerDEGPS_send : Real;
      RPMchanged : Bool;
      DirectionChanged : Bool;
      haltAxis : Bool;
   END_VAR
   VAR CONSTANT
      RollerMotorMaxSpeed : Real := 200.0;   // RPM
      MotorToRollerGearRatio : Real := 1.0;   // Belt transmission ratio
      RPMtoDEGSEC : Real := 6.0;   // RPM to Degress per Second conversion factor
      RollerDiameter : DInt := 50000;   // Diameter in microns
      LinearRollerSpeedFactor : Real;   // To convert rotation to linear speed
      RollerPWMPeriod : Int := 10000;
      RollerMinRPM : Real := 5.0;
   END_VAR
   // hscData.EnHSC := TRUE;
   // hscData.EnPeriod := false;
   // hscData.NewPeriod := 1000;
   VAR_TEMP   // added for the SCL form of the ladder/FBD networks
      _w1 : Bool;
      _w2 : Bool;
   END_VAR
BEGIN

REGION Network 1: Roller ON and Speed Control
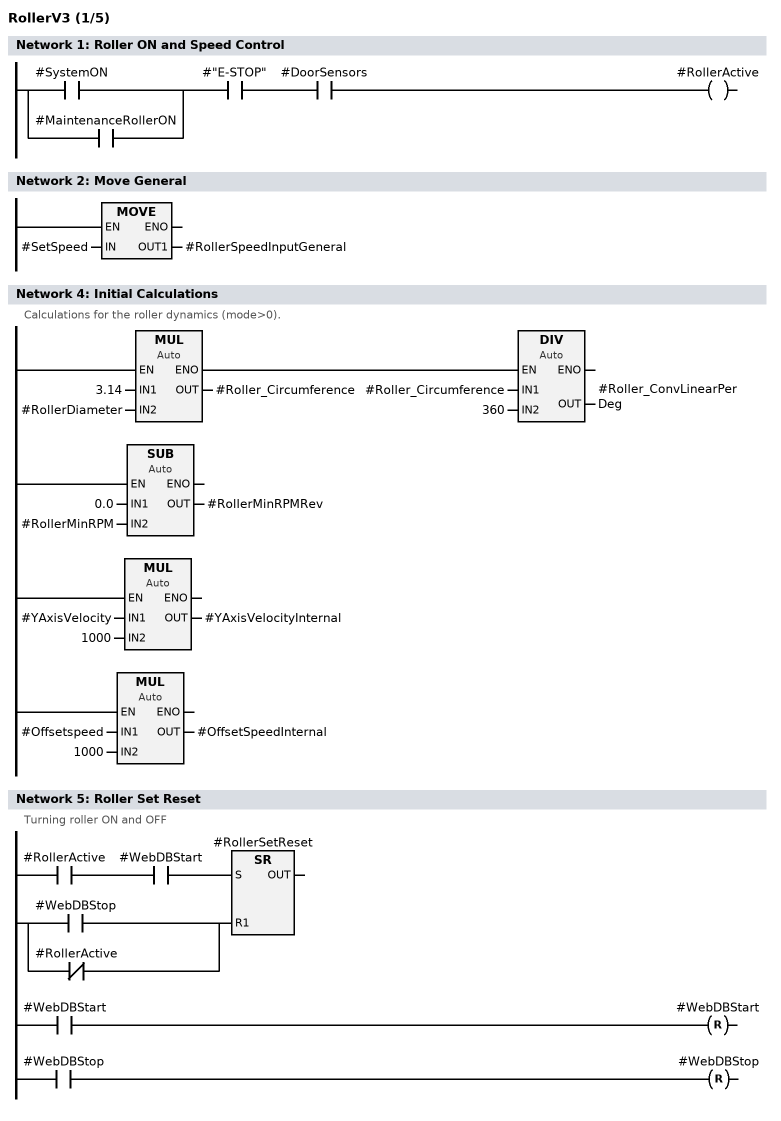
   RUNG wire#powerrail
      Contact( #SystemON )
      wire#w1
      Contact( #"E-STOP" )
      Contact( #DoorSensors )
      Coil( #RollerActive )
   END_RUNG
   RUNG wire#powerrail
      Contact( #MaintenanceRollerON )
   END_RUNG wire#w1
   // the same network as SCL:
   #RollerActive := (#SystemON OR #MaintenanceRollerON) AND #"E-STOP" AND #DoorSensors;
END_REGION

REGION Network 2: Move General
   RUNG wire#powerrail
      Move(in := #SetSpeed, out1 => #RollerSpeedInputGeneral)
   END_RUNG
   // the same network as SCL:
   #RollerSpeedInputGeneral := #SetSpeed;
END_REGION

REGION Network 3: Roller Direction
END_REGION

REGION Network 4: Initial Calculations
   // Calculations for the roller dynamics (mode>0).
   RUNG wire#powerrail
      Mul(in1 := 3.14, in2 := #RollerDiameter, out => #Roller_Circumference)
      Div(in1 := #Roller_Circumference, in2 := 360, out => #Roller_ConvLinearPerDeg)
   END_RUNG
   RUNG wire#powerrail
      Sub(in1 := 0.0, in2 := #RollerMinRPM, out => #RollerMinRPMRev)
   END_RUNG
   RUNG wire#powerrail
      Mul(in1 := #YAxisVelocity, in2 := 1000, out => #YAxisVelocityInternal)
   END_RUNG
   RUNG wire#powerrail
      Mul(in1 := #Offsetspeed, in2 := 1000, out => #OffsetSpeedInternal)
   END_RUNG
   // the same network as SCL:
   #Roller_Circumference := 3.14 * #RollerDiameter;
   #Roller_ConvLinearPerDeg := #Roller_Circumference / 360;
   #RollerMinRPMRev := 0.0 - #RollerMinRPM;
   #YAxisVelocityInternal := #YAxisVelocity * 1000;
   #OffsetSpeedInternal := #Offsetspeed * 1000;
END_REGION

REGION Network 5: Roller Set Reset
   // Turning roller ON and OFF
   RUNG wire#powerrail
      Contact( #RollerActive )
      Contact( #WebDBStart )
      S_SR(operand := #RollerSetReset, r1 := wire#w1)
   END_RUNG
   RUNG wire#powerrail
      Contact( #WebDBStop )
   END_RUNG wire#w1
   RUNG wire#powerrail
      I_Contact( #RollerActive )
   END_RUNG wire#w1
   RUNG wire#powerrail
      Contact( #WebDBStart )
      R_Coil( #WebDBStart )
   END_RUNG
   RUNG wire#powerrail
      Contact( #WebDBStop )
      R_Coil( #WebDBStop )
   END_RUNG
   // the same network as SCL:
   IF #RollerActive AND #WebDBStart THEN
       #RollerSetReset := TRUE;   // SR flip-flop
   END_IF;
   IF #WebDBStop OR NOT #RollerActive THEN #RollerSetReset := FALSE; END_IF;
   IF #WebDBStart THEN #WebDBStart := FALSE; END_IF;
   IF #WebDBStop THEN #WebDBStop := FALSE; END_IF;
END_REGION

REGION Network 6: PID
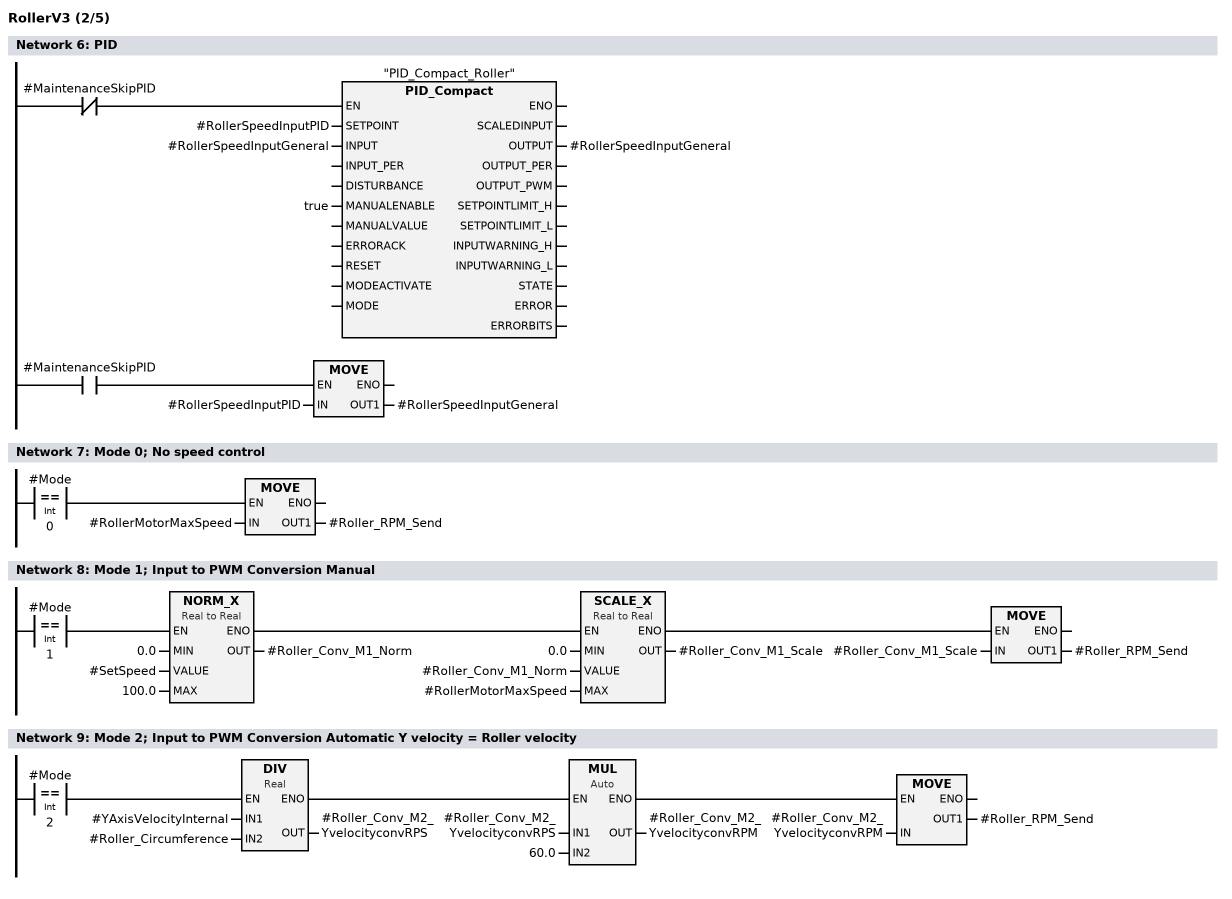
   RUNG wire#powerrail
      I_Contact( #MaintenanceSkipPID )
      "PID_Compact_Roller".PID_Compact(Setpoint := #RollerSpeedInputPID, Input := #RollerSpeedInputGeneral, Input_PER :=, Disturbance :=, ManualEnable := true, ManualValue :=, ErrorAck :=, Reset :=, ModeActivate :=, Mode :=, ScaledInput =>, Output => #RollerSpeedInputGeneral, Output_PER =>, Output_PWM =>, SetpointLimit_H =>, SetpointLimit_L =>, InputWarning_H =>, InputWarning_L =>, State =>, Error =>, ErrorBits =>)
   END_RUNG
   RUNG wire#powerrail
      Contact( #MaintenanceSkipPID )
      Move(in := #RollerSpeedInputPID, out1 => #RollerSpeedInputGeneral)
   END_RUNG
   // the same network as SCL:
   IF NOT #MaintenanceSkipPID THEN
       "PID_Compact_Roller"(Setpoint := #RollerSpeedInputPID,   // PID_Compact
                            Input := #RollerSpeedInputGeneral,
                            ManualEnable := true,
                            Output => #RollerSpeedInputGeneral);
   END_IF;
   IF #MaintenanceSkipPID THEN #RollerSpeedInputGeneral := #RollerSpeedInputPID; END_IF;
END_REGION

REGION Network 7: Mode 0; No speed control
   RUNG wire#powerrail
      { S7_Templates := "SrcType := Int" } EQ_Contact(in1 := #Mode, in2 := 0)
      Move(in := #RollerMotorMaxSpeed, out1 => #Roller_RPM_Send)
   END_RUNG
   // the same network as SCL:
   IF #Mode = 0 THEN #Roller_RPM_Send := #RollerMotorMaxSpeed; END_IF;
END_REGION

REGION Network 8: Mode 1; Input to PWM Conversion Manual
   RUNG wire#powerrail
      { S7_Templates := "SrcType := Int" } EQ_Contact(in1 := #Mode, in2 := 1)
      { S7_Templates := "[SrcType := Real, DestType := Real]" } Normalize(min := 0.0, value := #SetSpeed, max := 100.0, out => #Roller_Conv_M1_Norm)
      { S7_Templates := "[SrcType := Real, DestType := Real]" } Scale(min := 0.0, value := #Roller_Conv_M1_Norm, max := #RollerMotorMaxSpeed, out => #Roller_Conv_M1_Scale)
      Move(in := #Roller_Conv_M1_Scale, out1 => #Roller_RPM_Send)
   END_RUNG
   // the same network as SCL:
   IF #Mode = 1 THEN
       #Roller_Conv_M1_Norm := NORM_X(MIN := 0.0, VALUE := #SetSpeed, MAX := 100.0);
       #Roller_Conv_M1_Scale := SCALE_X(MIN := 0.0, VALUE := #Roller_Conv_M1_Norm, MAX := #RollerMotorMaxSpeed);
       #Roller_RPM_Send := #Roller_Conv_M1_Scale;
   END_IF;
END_REGION

REGION Network 9: Mode 2; Input to PWM Conversion Automatic Y velocity = Roller velocity
   RUNG wire#powerrail
      { S7_Templates := "SrcType := Int" } EQ_Contact(in1 := #Mode, in2 := 2)
      { S7_Templates := "SrcType := Real" } Div(in1 := #YAxisVelocityInternal, in2 := #Roller_Circumference, out => #Roller_Conv_M2_YvelocityconvRPS)
      Mul(in1 := #Roller_Conv_M2_YvelocityconvRPS, in2 := 60.0, out => #Roller_Conv_M2_YvelocityconvRPM)
      Move(in := #Roller_Conv_M2_YvelocityconvRPM, out1 => #Roller_RPM_Send)
   END_RUNG
   // the same network as SCL:
   IF #Mode = 2 THEN
       #Roller_Conv_M2_YvelocityconvRPS := #YAxisVelocityInternal / #Roller_Circumference;
       #Roller_Conv_M2_YvelocityconvRPM := #Roller_Conv_M2_YvelocityconvRPS * 60.0;
       #Roller_RPM_Send := #Roller_Conv_M2_YvelocityconvRPM;
   END_IF;
END_REGION

REGION Network 10: Mode 3; Input to PWM Conversion Setting Speed Difference according to the Y velocity
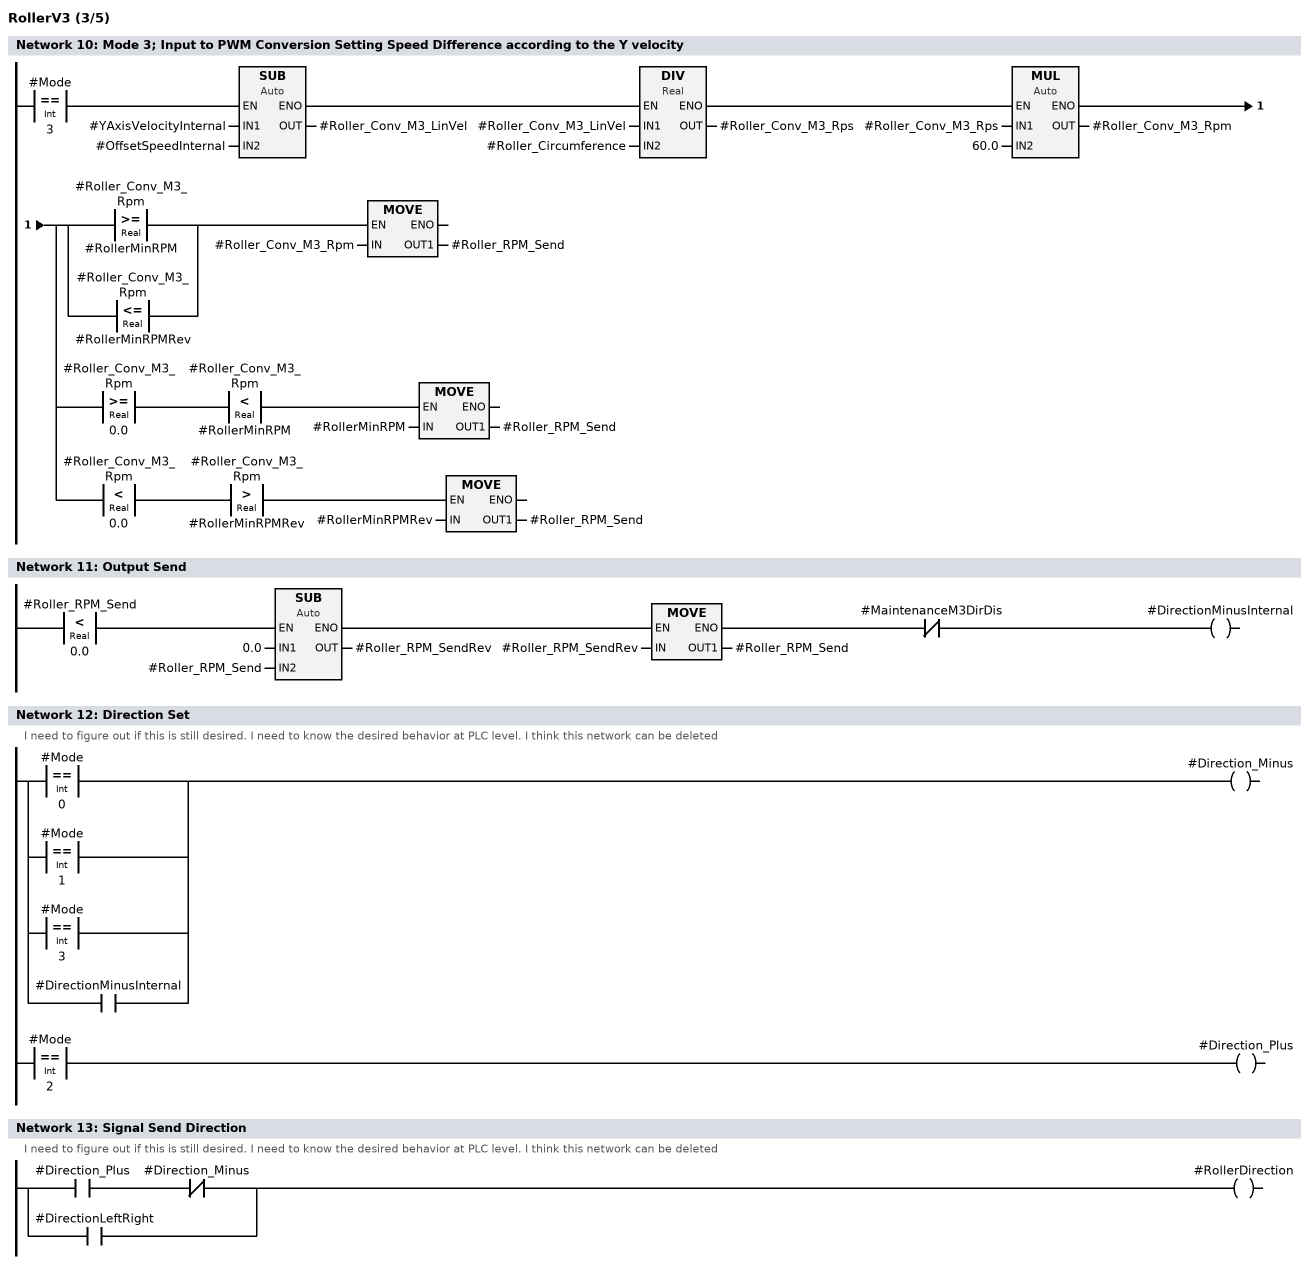
   RUNG wire#powerrail
      { S7_Templates := "SrcType := Int" } EQ_Contact(in1 := #Mode, in2 := 3)
      Sub(in1 := #YAxisVelocityInternal, in2 := #OffsetSpeedInternal, out => #Roller_Conv_M3_LinVel)
      { S7_Templates := "SrcType := Real" } Div(in1 := #Roller_Conv_M3_LinVel, in2 := #Roller_Circumference, out => #Roller_Conv_M3_Rps)
      Mul(in1 := #Roller_Conv_M3_Rps, in2 := 60.0, out => #Roller_Conv_M3_Rpm)
      wire#w1
      { S7_Templates := "SrcType := Real" } GE_Contact(in1 := #Roller_Conv_M3_Rpm, in2 := #RollerMinRPM)
      wire#w2
      Move(in := #Roller_Conv_M3_Rpm, out1 => #Roller_RPM_Send)
   END_RUNG
   RUNG wire#w1
      { S7_Templates := "SrcType := Real" } LE_Contact(in1 := #Roller_Conv_M3_Rpm, in2 := #RollerMinRPMRev)
   END_RUNG wire#w2
   RUNG wire#w1
      { S7_Templates := "SrcType := Real" } GE_Contact(in1 := #Roller_Conv_M3_Rpm, in2 := 0.0)
      { S7_Templates := "SrcType := Real" } LT_Contact(in1 := #Roller_Conv_M3_Rpm, in2 := #RollerMinRPM)
      Move(in := #RollerMinRPM, out1 => #Roller_RPM_Send)
   END_RUNG
   RUNG wire#w1
      { S7_Templates := "SrcType := Real" } LT_Contact(in1 := #Roller_Conv_M3_Rpm, in2 := 0.0)
      { S7_Templates := "SrcType := Real" } GT_Contact(in1 := #Roller_Conv_M3_Rpm, in2 := #RollerMinRPMRev)
      Move(in := #RollerMinRPMRev, out1 => #Roller_RPM_Send)
   END_RUNG
   // the same network as SCL:
   #_w1 := #Mode = 3;
   IF #_w1 THEN
       #Roller_Conv_M3_LinVel := #YAxisVelocityInternal - #OffsetSpeedInternal;
       #Roller_Conv_M3_Rps := #Roller_Conv_M3_LinVel / #Roller_Circumference;
       #Roller_Conv_M3_Rpm := #Roller_Conv_M3_Rps * 60.0;
   END_IF;
   IF #_w1 AND ((#Roller_Conv_M3_Rpm >= #RollerMinRPM) OR (#Roller_Conv_M3_Rpm <= #RollerMinRPMRev)) THEN
       #Roller_RPM_Send := #Roller_Conv_M3_Rpm;
   END_IF;
   IF #_w1 AND (#Roller_Conv_M3_Rpm >= 0.0) AND (#Roller_Conv_M3_Rpm < #RollerMinRPM) THEN
       #Roller_RPM_Send := #RollerMinRPM;
   END_IF;
   IF #_w1 AND (#Roller_Conv_M3_Rpm < 0.0) AND (#Roller_Conv_M3_Rpm > #RollerMinRPMRev) THEN
       #Roller_RPM_Send := #RollerMinRPMRev;
   END_IF;
END_REGION

REGION Network 11: Output Send
   RUNG wire#powerrail
      { S7_Templates := "SrcType := Real" } LT_Contact(in1 := #Roller_RPM_Send, in2 := 0.0)
      Sub(in1 := 0.0, in2 := #Roller_RPM_Send, out => #Roller_RPM_SendRev)
      Move(in := #Roller_RPM_SendRev, out1 => #Roller_RPM_Send)
      I_Contact( #MaintenanceM3DirDis )
      Coil( #DirectionMinusInternal )
   END_RUNG
   // the same network as SCL:
   #_w1 := #Roller_RPM_Send < 0.0;
   IF #_w1 THEN
       #Roller_RPM_SendRev := 0.0 - #Roller_RPM_Send;
       #Roller_RPM_Send := #Roller_RPM_SendRev;
   END_IF;
   #DirectionMinusInternal := #_w1 AND NOT #MaintenanceM3DirDis;
END_REGION

REGION Network 12: Direction Set
   // I need to figure out if this is still desired. I need to know the desired behavior at PLC level. I think this network can be deleted
   RUNG wire#powerrail
      { S7_Templates := "SrcType := Int" } EQ_Contact(in1 := #Mode, in2 := 0)
      wire#w1
      Coil( #Direction_Minus )
   END_RUNG
   RUNG wire#powerrail
      { S7_Templates := "SrcType := Int" } EQ_Contact(in1 := #Mode, in2 := 1)
   END_RUNG wire#w1
   RUNG wire#powerrail
      { S7_Templates := "SrcType := Int" } EQ_Contact(in1 := #Mode, in2 := 3)
   END_RUNG wire#w1
   RUNG wire#powerrail
      Contact( #DirectionMinusInternal )
   END_RUNG wire#w1
   RUNG wire#powerrail
      { S7_Templates := "SrcType := Int" } EQ_Contact(in1 := #Mode, in2 := 2)
      Coil( #Direction_Plus )
   END_RUNG
   // the same network as SCL:
   #Direction_Minus := (#Mode = 0) OR (#Mode = 1) OR (#Mode = 3) OR #DirectionMinusInternal;
   #Direction_Plus := #Mode = 2;
END_REGION

REGION Network 13: Signal Send Direction
   // I need to figure out if this is still desired. I need to know the desired behavior at PLC level. I think this network can be deleted
   RUNG wire#powerrail
      Contact( #Direction_Plus )
      I_Contact( #Direction_Minus )
      wire#w1
      Coil( #RollerDirection )
   END_RUNG
   RUNG wire#powerrail
      Contact( #DirectionLeftRight )
   END_RUNG wire#w1
   // the same network as SCL:
   #RollerDirection := (#Direction_Plus AND NOT #Direction_Minus) OR #DirectionLeftRight;
END_REGION

REGION Network 14
   // Convert Rotations per minute to degrees per second, as the technology object works with degrees. First, copy RPM send to an output variable, for output/logging purposes.
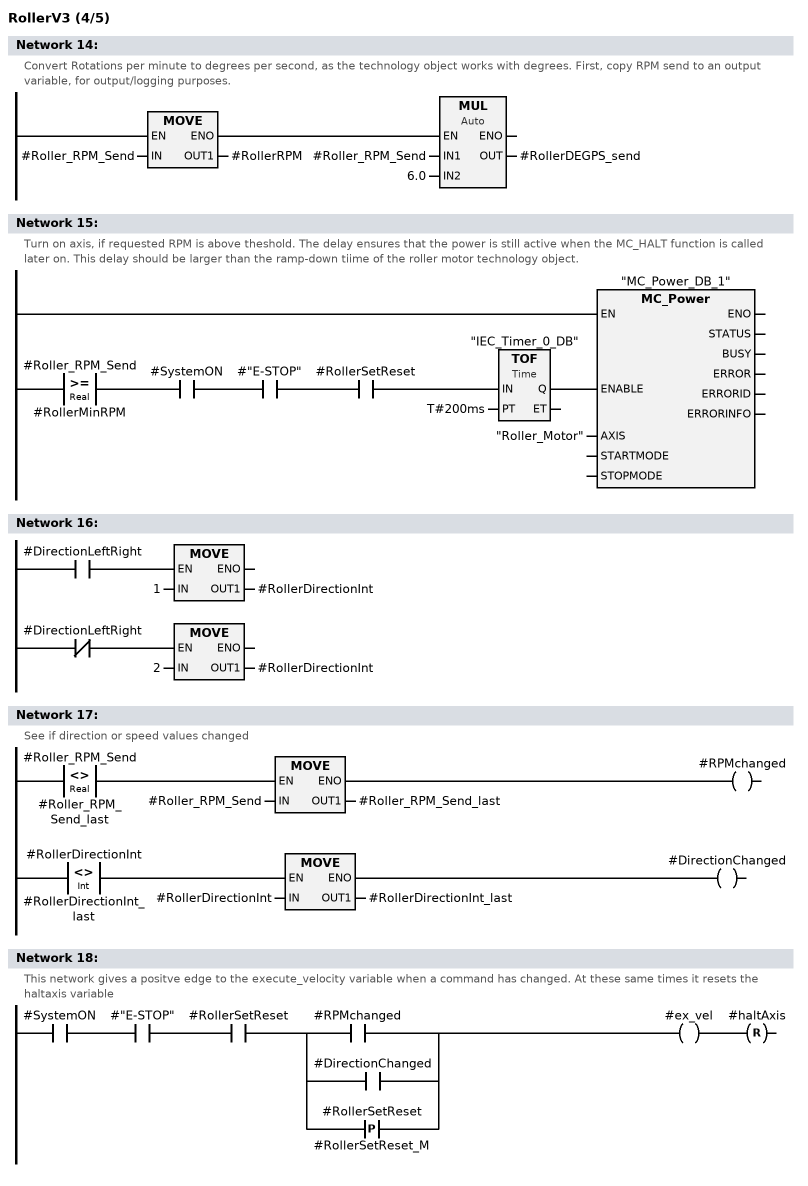
   RUNG wire#powerrail
      Move(in := #Roller_RPM_Send, out1 => #RollerRPM)
      Mul(in1 := #Roller_RPM_Send, in2 := 6.0, out => #RollerDEGPS_send)
   END_RUNG
   // the same network as SCL:
   #RollerRPM := #Roller_RPM_Send;
   #RollerDEGPS_send := #Roller_RPM_Send * 6.0;
END_REGION

REGION Network 15
   // Turn on axis, if requested RPM is above theshold. The delay ensures that the power is still active when the MC_HALT function is called later on. This delay should be larger than the ramp-down tiime of the roller motor technology object.
   RUNG wire#powerrail
      "MC_Power_DB_1".MC_Power(Enable := wire#w1, Axis := "Roller_Motor", StartMode :=, StopMode :=, Status =>, Busy =>, Error =>, ErrorID =>, ErrorInfo =>)
   END_RUNG
   RUNG wire#powerrail
      { S7_Templates := "SrcType := Real" } GE_Contact(in1 := #Roller_RPM_Send, in2 := #RollerMinRPM)
      Contact( #SystemON )
      Contact( #"E-STOP" )
      Contact( #RollerSetReset )
      { S7_Templates := "time_type := Time" } "IEC_Timer_0_DB".TOF(pt := T#200ms, et =>)
   END_RUNG wire#w1
   // the same network as SCL:
   "IEC_Timer_0_DB".TOF(IN := (#Roller_RPM_Send >= #RollerMinRPM) AND #SystemON AND #"E-STOP" AND #RollerSetReset,
                        PT := T#200ms);
   "MC_Power_DB_1"(Enable := "IEC_Timer_0_DB".Q, Axis := "Roller_Motor");   // MC_Power
END_REGION

REGION Network 16
   RUNG wire#powerrail
      Contact( #DirectionLeftRight )
      Move(in := 1, out1 => #RollerDirectionInt)
   END_RUNG
   RUNG wire#powerrail
      I_Contact( #DirectionLeftRight )
      Move(in := 2, out1 => #RollerDirectionInt)
   END_RUNG
   // the same network as SCL:
   IF #DirectionLeftRight THEN #RollerDirectionInt := 1; END_IF;
   IF NOT #DirectionLeftRight THEN #RollerDirectionInt := 2; END_IF;
END_REGION

REGION Network 17
   // See if direction or speed values changed
   RUNG wire#powerrail
      { S7_Templates := "SrcType := Real" } NE_Contact(in1 := #Roller_RPM_Send, in2 := #Roller_RPM_Send_last)
      Move(in := #Roller_RPM_Send, out1 => #Roller_RPM_Send_last)
      Coil( #RPMchanged )
   END_RUNG
   RUNG wire#powerrail
      { S7_Templates := "SrcType := Int" } NE_Contact(in1 := #RollerDirectionInt, in2 := #RollerDirectionInt_last)
      Move(in := #RollerDirectionInt, out1 => #RollerDirectionInt_last)
      Coil( #DirectionChanged )
   END_RUNG
   // the same network as SCL:
   #_w1 := #Roller_RPM_Send <> #Roller_RPM_Send_last;
   IF #_w1 THEN #Roller_RPM_Send_last := #Roller_RPM_Send; END_IF;
   #RPMchanged := #_w1;
   #_w2 := #RollerDirectionInt <> #RollerDirectionInt_last;
   IF #_w2 THEN #RollerDirectionInt_last := #RollerDirectionInt; END_IF;
   #DirectionChanged := #_w2;
END_REGION

REGION Network 18
   // This network gives a positve edge to the execute_velocity variable when a command has changed. At these same times it resets the haltaxis variable
   RUNG wire#powerrail
      Contact( #SystemON )
      Contact( #"E-STOP" )
      Contact( #RollerSetReset )
      wire#w1
      Contact( #RPMchanged )
      wire#w2
      Coil( #ex_vel )
      R_Coil( #haltAxis )
   END_RUNG
   RUNG wire#w1
      Contact( #DirectionChanged )
   END_RUNG wire#w2
   RUNG wire#w1
      P_Contact(operand := #RollerSetReset, bit := #RollerSetReset_M)
   END_RUNG wire#w2
   // the same network as SCL:
   #_w1 := #SystemON AND #"E-STOP" AND #RollerSetReset AND #RollerSetReset AND NOT #RollerSetReset_M;   // rising edge of #RollerSetReset
   #RollerSetReset_M := #RollerSetReset;
   #ex_vel := (#SystemON AND #"E-STOP" AND #RollerSetReset AND (#RPMchanged OR #DirectionChanged)) OR #_w1;
   IF #ex_vel THEN #haltAxis := FALSE; END_IF;
END_REGION

REGION Network 19: Convert dircetion command to INT; Send command to drive
   // Direction; 0 means that the direction is in the sigh of the velocity; 1 is positive direction; 2 is negative direction
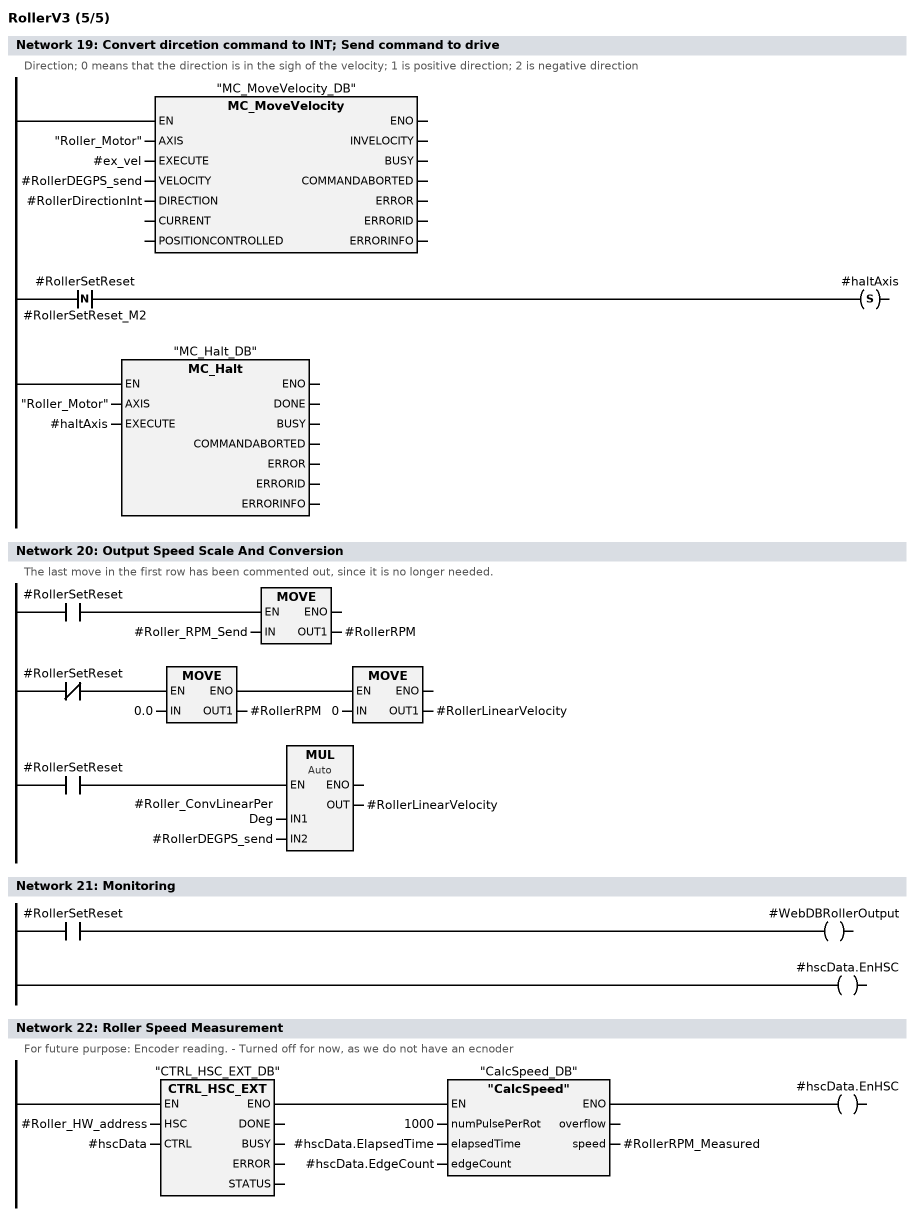
   RUNG wire#powerrail
      "MC_MoveVelocity_DB".MC_MoveVelocity(Axis := "Roller_Motor", Execute := #ex_vel, Velocity := #RollerDEGPS_send, Direction := #RollerDirectionInt, Current :=, PositionControlled :=, InVelocity =>, Busy =>, CommandAborted =>, Error =>, ErrorID =>, ErrorInfo =>)
   END_RUNG
   RUNG wire#powerrail
      N_Contact(operand := #RollerSetReset, bit := #RollerSetReset_M2)
      S_Coil( #haltAxis )
   END_RUNG
   RUNG wire#powerrail
      "MC_Halt_DB".MC_Halt(Axis := "Roller_Motor", Execute := #haltAxis, Done =>, Busy =>, CommandAborted =>, Error =>, ErrorID =>, ErrorInfo =>)
   END_RUNG
   // the same network as SCL:
   "MC_MoveVelocity_DB"(Axis := "Roller_Motor",   // MC_MoveVelocity
                        Execute := #ex_vel,
                        Velocity := #RollerDEGPS_send,
                        Direction := #RollerDirectionInt);
   #_w1 := NOT #RollerSetReset AND #RollerSetReset_M2;   // falling edge of #RollerSetReset
   #RollerSetReset_M2 := #RollerSetReset;
   IF #_w1 THEN #haltAxis := TRUE; END_IF;
   "MC_Halt_DB"(Axis := "Roller_Motor", Execute := #haltAxis);   // MC_Halt
END_REGION

REGION Network 20: Output Speed Scale And Conversion
   // The last move in the first row has been commented out, since it is no longer needed.
   RUNG wire#powerrail
      Contact( #RollerSetReset )
      Move(in := #Roller_RPM_Send, out1 => #RollerRPM)
   END_RUNG
   RUNG wire#powerrail
      I_Contact( #RollerSetReset )
      Move(in := 0.0, out1 => #RollerRPM)
      Move(in := 0, out1 => #RollerLinearVelocity)
   END_RUNG
   RUNG wire#powerrail
      Contact( #RollerSetReset )
      Mul(in1 := #Roller_ConvLinearPerDeg, in2 := #RollerDEGPS_send, out => #RollerLinearVelocity)
   END_RUNG
   // the same network as SCL:
   IF #RollerSetReset THEN #RollerRPM := #Roller_RPM_Send; END_IF;
   IF NOT #RollerSetReset THEN
       #RollerRPM := 0.0;
       #RollerLinearVelocity := 0;
   END_IF;
   IF #RollerSetReset THEN #RollerLinearVelocity := #Roller_ConvLinearPerDeg * #RollerDEGPS_send; END_IF;
END_REGION

REGION Network 21: Monitoring
   RUNG wire#powerrail
      Contact( #RollerSetReset )
      Coil( #WebDBRollerOutput )
   END_RUNG
   RUNG wire#powerrail
      Coil( #hscData.EnHSC )
   END_RUNG
   // the same network as SCL:
   #WebDBRollerOutput := #RollerSetReset;
   #hscData.EnHSC := TRUE;
END_REGION

REGION Network 22: Roller Speed Measurement
   // For future purpose: Encoder reading. - Turned off for now, as we do not have an ecnoder
   RUNG wire#powerrail
      "CTRL_HSC_EXT_DB".CTRL_HSC_EXT(HSC := #Roller_HW_address, CTRL := #hscData, DONE =>, BUSY =>, ERROR =>, STATUS =>)
      "CalcSpeed_DB"(numPulsePerRot := 1000, elapsedTime := #hscData.ElapsedTime, edgeCount := #hscData.EdgeCount, overflow =>, speed => #RollerRPM_Measured)
      Coil( #hscData.EnHSC )
   END_RUNG
   // the same network as SCL:
   "CTRL_HSC_EXT_DB"(HSC := #Roller_HW_address, CTRL := #hscData, ENO => #_w1);   // CTRL_HSC_EXT
   "CalcSpeed_DB"(EN := #_w1,   // "CalcSpeed"
                  numPulsePerRot := 1000,
                  elapsedTime := #hscData.ElapsedTime,
                  edgeCount := #hscData.EdgeCount,
                  speed => #RollerRPM_Measured,
                  ENO => #_w2);
   #hscData.EnHSC := #_w2;
END_REGION
END_FUNCTION_BLOCK

FUNCTION_BLOCK "Z axis missing layer detection"   // FB3, LAD
TITLE = Description:
{ S7_Optimized_Access := 'TRUE' }
VERSION : 0.1
// Still in the development mode, not yet fully working.
// 
// Function block used to actively check if the positions of the Z1, Z2 axes are correct while printing. Missing layer detection is based on the check sum.
   VAR_INPUT
      Mode : DInt;
      PrintStarted : Bool;
      PrintPaused : Bool;
      PrintEnded : Bool;
      Z1AxisPosition : DInt;
      Z1FeedStep : DInt;
      Z1Relative : Bool;
      Z2AxisPosition : DInt;
      Z2StepSize : DInt;
      Z2Relative : Bool;
      AmountOfLayers : DInt := 100;
      MotionMargin : DInt := 5;
      CompensationStepSize : DInt := 500;
      PrintingStepSize : DInt := 100;
   END_VAR
   VAR_OUTPUT
      Z1PredictedFinalPositionMinus : DInt;
      Z1PredictedFinalPosition : DInt;
      Z1PredictedFinalPositionPlus : DInt;
      Z2PredictedFinalPositionMinus : DInt;
      Z2PredictedFinalPosition : DInt;
      Z2PredictedFinalPositionPlus : DInt;
      MissingLayerStatus : Bool;   // 0 if the print is fine; 1 if the layer was skipped
      ErrorTime : Time;
   END_VAR
   VAR
      CheckSumStart : DInt;
      CheckSumMarginPlus : DInt;
      CheckSumMarginMinus : DInt;
      CheckSumActual : DInt;
      MachinePrintingInternal : Bool;
      MachinePrintingInternalM1 : Bool;
      Z1StartPosition : DInt;
      Z2StartPosition : DInt;
      Z1AddedDistanceInternal : DInt;
      Z2AddedDistanceInternal : DInt;
   END_VAR
   VAR_TEMP   // added for the SCL form of the ladder/FBD networks
      _w1 : Bool;
   END_VAR
BEGIN

REGION Network 1: Machine Printing Status
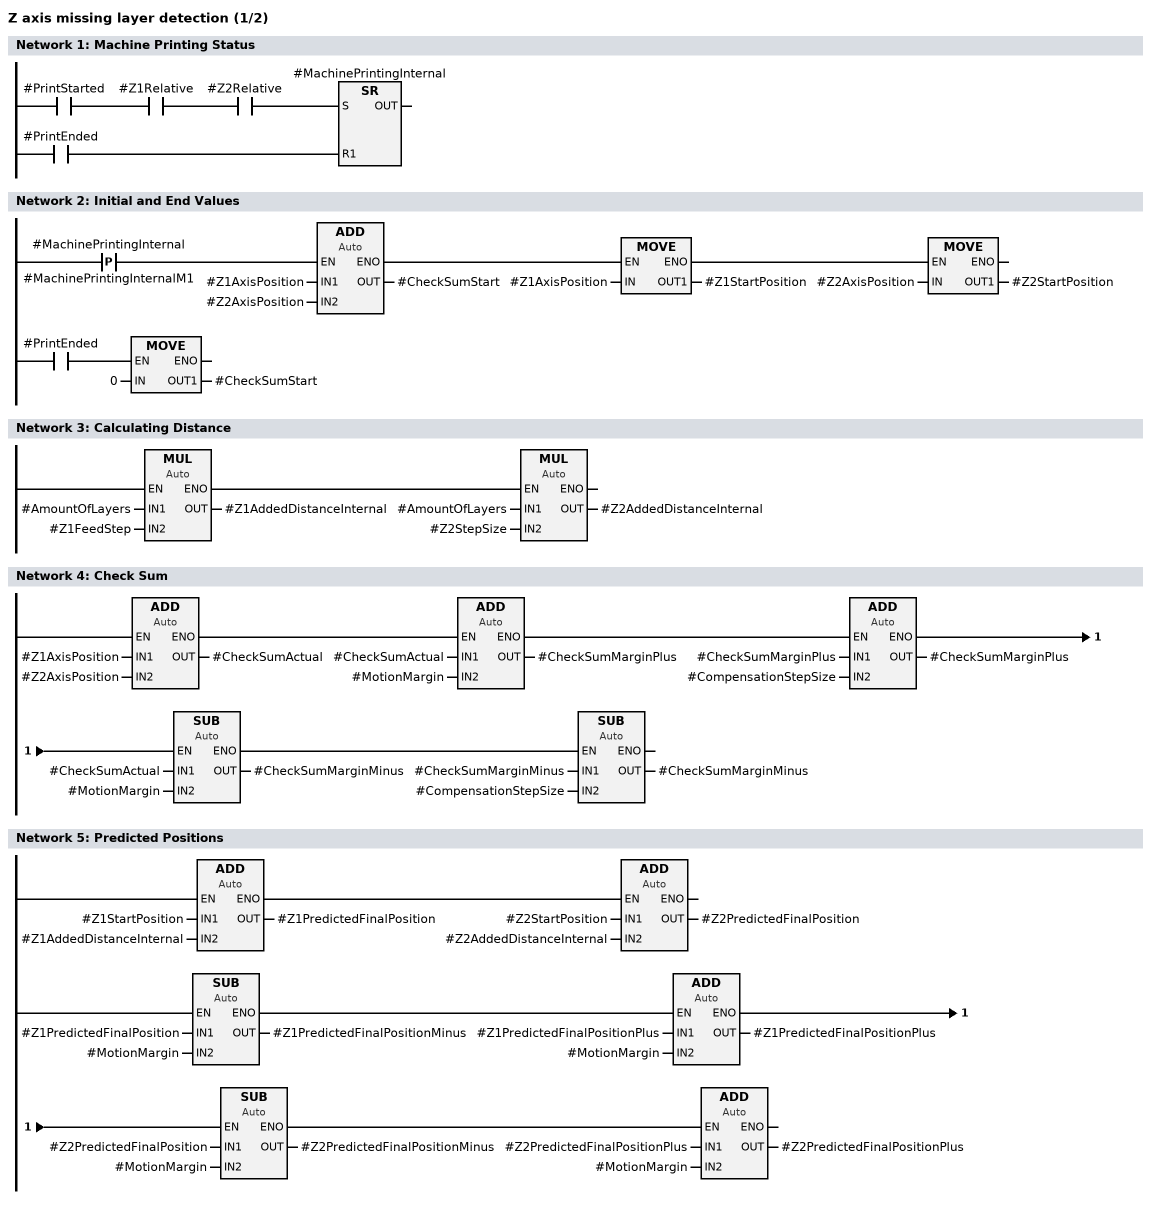
   RUNG wire#powerrail
      Contact( #PrintStarted )
      Contact( #Z1Relative )
      Contact( #Z2Relative )
      S_SR(operand := #MachinePrintingInternal, r1 := wire#w1)
   END_RUNG
   RUNG wire#powerrail
      Contact( #PrintEnded )
   END_RUNG wire#w1
   // the same network as SCL:
   IF #PrintStarted AND #Z1Relative AND #Z2Relative THEN
       #MachinePrintingInternal := TRUE;   // SR flip-flop
   END_IF;
   IF #PrintEnded THEN #MachinePrintingInternal := FALSE; END_IF;
END_REGION

REGION Network 2: Initial and End Values
   RUNG wire#powerrail
      P_Contact(operand := #MachinePrintingInternal, bit := #MachinePrintingInternalM1)
      Add(in1 := #Z1AxisPosition, in2 := #Z2AxisPosition, out => #CheckSumStart)
      Move(in := #Z1AxisPosition, out1 => #Z1StartPosition)
      Move(in := #Z2AxisPosition, out1 => #Z2StartPosition)
   END_RUNG
   RUNG wire#powerrail
      Contact( #PrintEnded )
      Move(in := 0, out1 => #CheckSumStart)
   END_RUNG
   // the same network as SCL:
   #_w1 := #MachinePrintingInternal AND NOT #MachinePrintingInternalM1;   // rising edge of #MachinePrintingInternal
   #MachinePrintingInternalM1 := #MachinePrintingInternal;
   IF #_w1 THEN
       #CheckSumStart := #Z1AxisPosition + #Z2AxisPosition;
       #Z1StartPosition := #Z1AxisPosition;
       #Z2StartPosition := #Z2AxisPosition;
   END_IF;
   IF #PrintEnded THEN #CheckSumStart := 0; END_IF;
END_REGION

REGION Network 3: Calculating Distance
   RUNG wire#powerrail
      Mul(in1 := #AmountOfLayers, in2 := #Z1FeedStep, out => #Z1AddedDistanceInternal)
      Mul(in1 := #AmountOfLayers, in2 := #Z2StepSize, out => #Z2AddedDistanceInternal)
   END_RUNG
   // the same network as SCL:
   #Z1AddedDistanceInternal := #AmountOfLayers * #Z1FeedStep;
   #Z2AddedDistanceInternal := #AmountOfLayers * #Z2StepSize;
END_REGION

REGION Network 4: Check Sum
   RUNG wire#powerrail
      Add(in1 := #Z1AxisPosition, in2 := #Z2AxisPosition, out => #CheckSumActual)
      Add(in1 := #CheckSumActual, in2 := #MotionMargin, out => #CheckSumMarginPlus)
      Add(in1 := #CheckSumMarginPlus, in2 := #CompensationStepSize, out => #CheckSumMarginPlus)
      Sub(in1 := #CheckSumActual, in2 := #MotionMargin, out => #CheckSumMarginMinus)
      Sub(in1 := #CheckSumMarginMinus, in2 := #CompensationStepSize, out => #CheckSumMarginMinus)
   END_RUNG
   // the same network as SCL:
   #CheckSumActual := #Z1AxisPosition + #Z2AxisPosition;
   #CheckSumMarginPlus := #CheckSumActual + #MotionMargin;
   #CheckSumMarginPlus := #CheckSumMarginPlus + #CompensationStepSize;
   #CheckSumMarginMinus := #CheckSumActual - #MotionMargin;
   #CheckSumMarginMinus := #CheckSumMarginMinus - #CompensationStepSize;
END_REGION

REGION Network 5: Predicted Positions
   RUNG wire#powerrail
      Add(in1 := #Z1StartPosition, in2 := #Z1AddedDistanceInternal, out => #Z1PredictedFinalPosition)
      Add(in1 := #Z2StartPosition, in2 := #Z2AddedDistanceInternal, out => #Z2PredictedFinalPosition)
   END_RUNG
   RUNG wire#powerrail
      Sub(in1 := #Z1PredictedFinalPosition, in2 := #MotionMargin, out => #Z1PredictedFinalPositionMinus)
      Add(in1 := #Z1PredictedFinalPositionPlus, in2 := #MotionMargin, out => #Z1PredictedFinalPositionPlus)
      Sub(in1 := #Z2PredictedFinalPosition, in2 := #MotionMargin, out => #Z2PredictedFinalPositionMinus)
      Add(in1 := #Z2PredictedFinalPositionPlus, in2 := #MotionMargin, out => #Z2PredictedFinalPositionPlus)
   END_RUNG
   // the same network as SCL:
   #Z1PredictedFinalPosition := #Z1StartPosition + #Z1AddedDistanceInternal;
   #Z2PredictedFinalPosition := #Z2StartPosition + #Z2AddedDistanceInternal;
   #Z1PredictedFinalPositionMinus := #Z1PredictedFinalPosition - #MotionMargin;
   #Z1PredictedFinalPositionPlus := #Z1PredictedFinalPositionPlus + #MotionMargin;
   #Z2PredictedFinalPositionMinus := #Z2PredictedFinalPosition - #MotionMargin;
   #Z2PredictedFinalPositionPlus := #Z2PredictedFinalPositionPlus + #MotionMargin;
END_REGION

REGION Network 6: Status
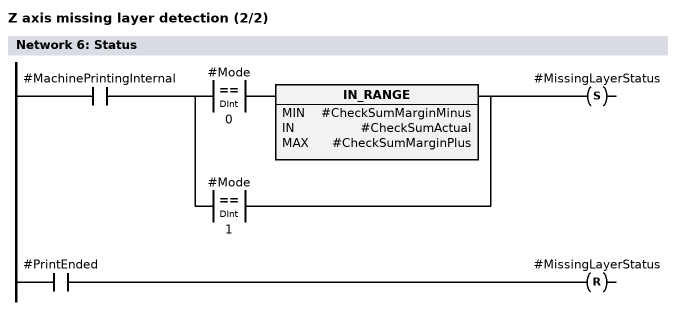
   RUNG wire#powerrail
      Contact( #MachinePrintingInternal )
      wire#w1
      { S7_Templates := "SrcType := DInt" } EQ_Contact(in1 := #Mode, in2 := 0)
      { S7_Templates := "SrcType := DInt" } InRange(min := #CheckSumMarginMinus, in := #CheckSumActual, max := #CheckSumMarginPlus)
      wire#w2
      S_Coil( #MissingLayerStatus )
   END_RUNG
   RUNG wire#w1
      { S7_Templates := "SrcType := DInt" } EQ_Contact(in1 := #Mode, in2 := 1)
   END_RUNG wire#w2
   RUNG wire#powerrail
      Contact( #PrintEnded )
      R_Coil( #MissingLayerStatus )
   END_RUNG
   // the same network as SCL:
   IF #MachinePrintingInternal AND (((#Mode = 0) AND (#CheckSumMarginMinus <= #CheckSumActual) AND (#CheckSumActual <= #CheckSumMarginPlus)) OR (#Mode = 1)) THEN
       #MissingLayerStatus := TRUE;
   END_IF;
   IF #PrintEnded THEN #MissingLayerStatus := FALSE; END_IF;
END_REGION
END_FUNCTION_BLOCK

FUNCTION_BLOCK "BOOL_DEMUX"   // FB13, LAD
{ S7_Optimized_Access := 'TRUE' }
VERSION : 0.1
   VAR_INPUT
      State : Int;
      Reset_cmd : Bool;
      Homing_all_axis : Bool;
   END_VAR
   VAR_OUTPUT
      Out1 : Bool;
      Out2 : Bool;
      Out3 : Bool;
      Out4 : Bool;
      Out5 : Bool;
      Out6 : Int;
   END_VAR
   VAR
      Edge_S_Out1 : Bool;
      Edge_M_Out1 : Bool;
      Edge_S_Out2 : Bool;
      Edge_M_Out2 : Bool;
      Edge_S_Out3 : Bool;
      Edge_M_Out3 : Bool;
      Edge_S_Out4 : Bool;
      Edge_M_Out4 : Bool;
      Edge_S_Out5 : Bool;
      Edge_M_Out5 : Bool;
   END_VAR
   VAR_TEMP   // added for the SCL form of the ladder/FBD networks
      _w1 : Bool;
   END_VAR
BEGIN

REGION Network 1
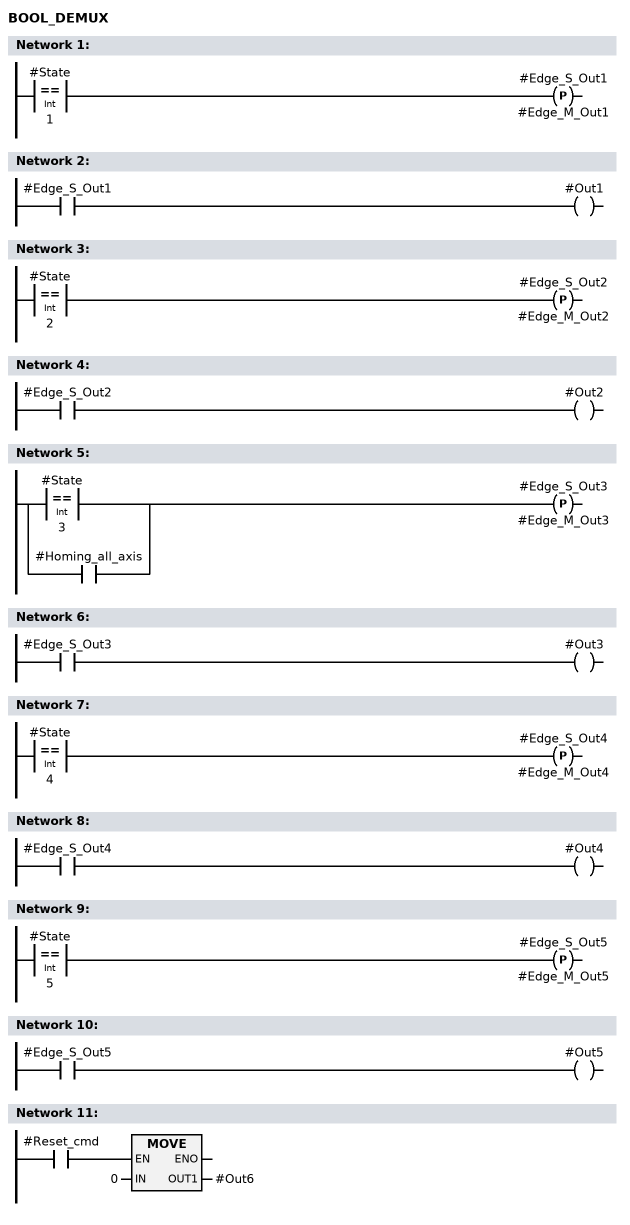
   #_w1 := #State = 1;
   #Edge_S_Out1 := #_w1 AND NOT #Edge_M_Out1;   // rising edge
   #Edge_M_Out1 := #_w1;
END_REGION

REGION Network 2
   RUNG wire#powerrail
      Contact( #Edge_S_Out1 )
      Coil( #Out1 )
   END_RUNG
   // the same network as SCL:
   #Out1 := #Edge_S_Out1;
END_REGION

REGION Network 3
   #_w1 := #State = 2;
   #Edge_S_Out2 := #_w1 AND NOT #Edge_M_Out2;   // rising edge
   #Edge_M_Out2 := #_w1;
END_REGION

REGION Network 4
   RUNG wire#powerrail
      Contact( #Edge_S_Out2 )
      Coil( #Out2 )
   END_RUNG
   // the same network as SCL:
   #Out2 := #Edge_S_Out2;
END_REGION

REGION Network 5
   #_w1 := (#State = 3) OR #Homing_all_axis;
   #Edge_S_Out3 := #_w1 AND NOT #Edge_M_Out3;   // rising edge
   #Edge_M_Out3 := #_w1;
END_REGION

REGION Network 6
   RUNG wire#powerrail
      Contact( #Edge_S_Out3 )
      Coil( #Out3 )
   END_RUNG
   // the same network as SCL:
   #Out3 := #Edge_S_Out3;
END_REGION

REGION Network 7
   #_w1 := #State = 4;
   #Edge_S_Out4 := #_w1 AND NOT #Edge_M_Out4;   // rising edge
   #Edge_M_Out4 := #_w1;
END_REGION

REGION Network 8
   RUNG wire#powerrail
      Contact( #Edge_S_Out4 )
      Coil( #Out4 )
   END_RUNG
   // the same network as SCL:
   #Out4 := #Edge_S_Out4;
END_REGION

REGION Network 9
   #_w1 := #State = 5;
   #Edge_S_Out5 := #_w1 AND NOT #Edge_M_Out5;   // rising edge
   #Edge_M_Out5 := #_w1;
END_REGION

REGION Network 10
   RUNG wire#powerrail
      Contact( #Edge_S_Out5 )
      Coil( #Out5 )
   END_RUNG
   // the same network as SCL:
   #Out5 := #Edge_S_Out5;
END_REGION

REGION Network 11
   RUNG wire#powerrail
      Contact( #Reset_cmd )
      Move(in := 0, out1 => #Out6)
   END_RUNG
   // the same network as SCL:
   IF #Reset_cmd THEN #Out6 := 0; END_IF;
END_REGION
END_FUNCTION_BLOCK

FUNCTION "DevTempGarb" : Void   // FC13, LAD
TITLE = Development garbarge area
{ S7_Optimized_Access := 'TRUE' }
AUTHOR : HenriP
VERSION : 0.1
// To use when removing part of the code for test
BEGIN
END_FUNCTION

FUNCTION "MainDevTrashBin" : Void   // FC17, LAD
{ S7_Optimized_Access := 'TRUE' }
AUTHOR : HenriP
VERSION : 0.1
   VAR_TEMP
      AxisFault : Bool;
   END_VAR
BEGIN

REGION Network 2: Initial step
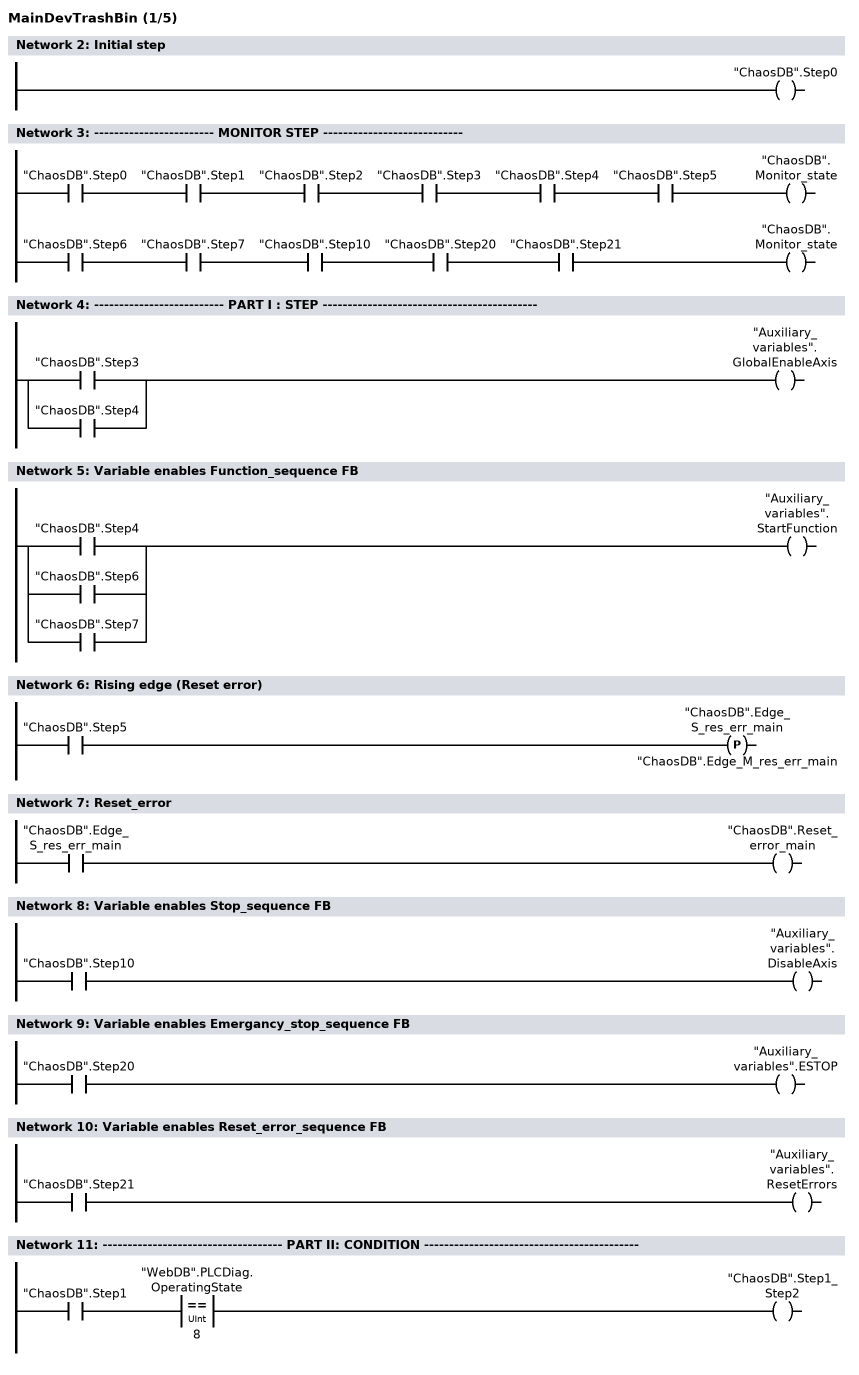
   RUNG wire#powerrail
      Coil( "ChaosDB".Step0 )
   END_RUNG
   // the same network as SCL:
   "ChaosDB".Step0 := TRUE;
END_REGION

REGION Network 3: ------------------------ MONITOR STEP ----------------------------
   RUNG wire#powerrail
      Contact( "ChaosDB".Step0 )
      Contact( "ChaosDB".Step1 )
      Contact( "ChaosDB".Step2 )
      Contact( "ChaosDB".Step3 )
      Contact( "ChaosDB".Step4 )
      Contact( "ChaosDB".Step5 )
      Coil( "ChaosDB".Monitor_state )
   END_RUNG
   RUNG wire#powerrail
      Contact( "ChaosDB".Step6 )
      Contact( "ChaosDB".Step7 )
      Contact( "ChaosDB".Step10 )
      Contact( "ChaosDB".Step20 )
      Contact( "ChaosDB".Step21 )
      Coil( "ChaosDB".Monitor_state )
   END_RUNG
   // the same network as SCL:
   "ChaosDB".Monitor_state := "ChaosDB".Step0 AND "ChaosDB".Step1 AND "ChaosDB".Step2 AND "ChaosDB".Step3 AND "ChaosDB".Step4 AND "ChaosDB".Step5;
   "ChaosDB".Monitor_state := "ChaosDB".Step6 AND "ChaosDB".Step7 AND "ChaosDB".Step10 AND "ChaosDB".Step20 AND "ChaosDB".Step21;
END_REGION

REGION Network 4: -------------------------- PART I : STEP -------------------------------------------
   RUNG wire#powerrail
      Contact( "ChaosDB".Step3 )
      wire#w1
      Coil( "Auxiliary_variables".GlobalEnableAxis )
   END_RUNG
   RUNG wire#powerrail
      Contact( "ChaosDB".Step4 )
   END_RUNG wire#w1
   // the same network as SCL:
   "Auxiliary_variables".GlobalEnableAxis := "ChaosDB".Step3 OR "ChaosDB".Step4;
END_REGION

REGION Network 5: Variable enables Function_sequence FB
   RUNG wire#powerrail
      Contact( "ChaosDB".Step4 )
      wire#w1
      Coil( "Auxiliary_variables".StartFunction )
   END_RUNG
   RUNG wire#powerrail
      Contact( "ChaosDB".Step6 )
   END_RUNG wire#w1
   RUNG wire#powerrail
      Contact( "ChaosDB".Step7 )
   END_RUNG wire#w1
   // the same network as SCL:
   "Auxiliary_variables".StartFunction := "ChaosDB".Step4 OR "ChaosDB".Step6 OR "ChaosDB".Step7;
END_REGION

REGION Network 6: Rising edge (Reset error)
   "ChaosDB".Edge_S_res_err_main := "ChaosDB".Step5 AND NOT "ChaosDB".Edge_M_res_err_main;   // rising edge
   "ChaosDB".Edge_M_res_err_main := "ChaosDB".Step5;
END_REGION

REGION Network 7: Reset_error
   RUNG wire#powerrail
      Contact( "ChaosDB".Edge_S_res_err_main )
      Coil( "ChaosDB".Reset_error_main )
   END_RUNG
   // the same network as SCL:
   "ChaosDB".Reset_error_main := "ChaosDB".Edge_S_res_err_main;
END_REGION

REGION Network 8: Variable enables Stop_sequence FB
   RUNG wire#powerrail
      Contact( "ChaosDB".Step10 )
      Coil( "Auxiliary_variables".DisableAxis )
   END_RUNG
   // the same network as SCL:
   "Auxiliary_variables".DisableAxis := "ChaosDB".Step10;
END_REGION

REGION Network 9: Variable enables Emergancy_stop_sequence FB
   RUNG wire#powerrail
      Contact( "ChaosDB".Step20 )
      Coil( "Auxiliary_variables".ESTOP )
   END_RUNG
   // the same network as SCL:
   "Auxiliary_variables".ESTOP := "ChaosDB".Step20;
END_REGION

REGION Network 10: Variable enables Reset_error_sequence FB
   RUNG wire#powerrail
      Contact( "ChaosDB".Step21 )
      Coil( "Auxiliary_variables".ResetErrors )
   END_RUNG
   // the same network as SCL:
   "Auxiliary_variables".ResetErrors := "ChaosDB".Step21;
END_REGION

REGION Network 11: ------------------------------------ PART II: CONDITION -------------------------------------------
   RUNG wire#powerrail
      Contact( "ChaosDB".Step1 )
      { S7_Templates := "SrcType := UInt" } EQ_Contact(in1 := "WebDB".PLCDiag.OperatingState, in2 := 8)
      Coil( "ChaosDB".Step1_Step2 )
   END_RUNG
   // the same network as SCL:
   "ChaosDB".Step1_Step2 := "ChaosDB".Step1 AND ("WebDB".PLCDiag.OperatingState = 8);
END_REGION

REGION Network 12
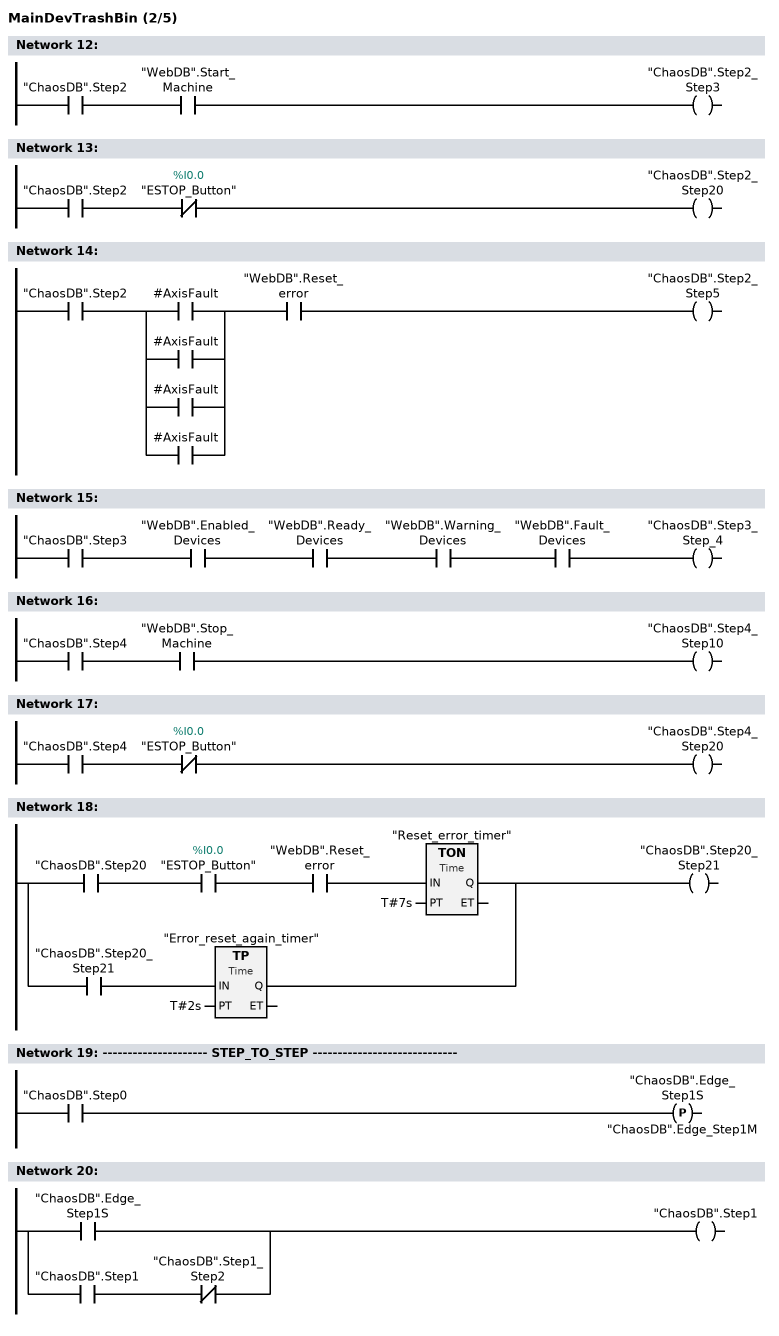
   RUNG wire#powerrail
      Contact( "ChaosDB".Step2 )
      Contact( "WebDB".Start_Machine )
      Coil( "ChaosDB".Step2_Step3 )
   END_RUNG
   // the same network as SCL:
   "ChaosDB".Step2_Step3 := "ChaosDB".Step2 AND "WebDB".Start_Machine;
END_REGION

REGION Network 13
   RUNG wire#powerrail
      Contact( "ChaosDB".Step2 )
      I_Contact( "ESTOP_Button" )
      Coil( "ChaosDB".Step2_Step20 )
   END_RUNG
   // the same network as SCL:
   "ChaosDB".Step2_Step20 := "ChaosDB".Step2 AND NOT "ESTOP_Button";
END_REGION

REGION Network 14
   RUNG wire#powerrail
      Contact( "ChaosDB".Step2 )
      wire#w1
      Contact( #AxisFault )
      wire#w2
      Contact( "WebDB".Reset_error )
      Coil( "ChaosDB".Step2_Step5 )
   END_RUNG
   RUNG wire#w1
      Contact( #AxisFault )
   END_RUNG wire#w2
   RUNG wire#w1
      Contact( #AxisFault )
   END_RUNG wire#w2
   RUNG wire#w1
      Contact( #AxisFault )
   END_RUNG wire#w2
   // the same network as SCL:
   "ChaosDB".Step2_Step5 := "ChaosDB".Step2 AND (#AxisFault OR #AxisFault OR #AxisFault OR #AxisFault) AND "WebDB".Reset_error;
END_REGION

REGION Network 15
   RUNG wire#powerrail
      Contact( "ChaosDB".Step3 )
      Contact( "WebDB".Enabled_Devices )
      Contact( "WebDB".Ready_Devices )
      Contact( "WebDB".Warning_Devices )
      Contact( "WebDB".Fault_Devices )
      Coil( "ChaosDB".Step3_Step_4 )
   END_RUNG
   // the same network as SCL:
   "ChaosDB".Step3_Step_4 := "ChaosDB".Step3 AND "WebDB".Enabled_Devices AND "WebDB".Ready_Devices AND "WebDB".Warning_Devices AND "WebDB".Fault_Devices;
END_REGION

REGION Network 16
   RUNG wire#powerrail
      Contact( "ChaosDB".Step4 )
      Contact( "WebDB".Stop_Machine )
      Coil( "ChaosDB".Step4_Step10 )
   END_RUNG
   // the same network as SCL:
   "ChaosDB".Step4_Step10 := "ChaosDB".Step4 AND "WebDB".Stop_Machine;
END_REGION

REGION Network 17
   RUNG wire#powerrail
      Contact( "ChaosDB".Step4 )
      I_Contact( "ESTOP_Button" )
      Coil( "ChaosDB".Step4_Step20 )
   END_RUNG
   // the same network as SCL:
   "ChaosDB".Step4_Step20 := "ChaosDB".Step4 AND NOT "ESTOP_Button";
END_REGION

REGION Network 18
   RUNG wire#powerrail
      Contact( "ChaosDB".Step20 )
      Contact( "ESTOP_Button" )
      Contact( "WebDB".Reset_error )
      { S7_Templates := "time_type := Time" } "Reset_error_timer".TON(pt := T#7s, et =>)
      wire#w1
      Coil( "ChaosDB".Step20_Step21 )
   END_RUNG
   RUNG wire#powerrail
      Contact( "ChaosDB".Step20_Step21 )
      { S7_Templates := "time_type := Time" } "Error_reset_again_timer".TP(pt := T#2s, et =>)
   END_RUNG wire#w1
   // the same network as SCL:
   "Reset_error_timer".TON(IN := "ChaosDB".Step20 AND "ESTOP_Button" AND "WebDB".Reset_error, PT := T#7s);
   "Error_reset_again_timer".TP(IN := "ChaosDB".Step20_Step21, PT := T#2s);
   "ChaosDB".Step20_Step21 := "Reset_error_timer".Q OR "Error_reset_again_timer".Q;
END_REGION

REGION Network 19: --------------------- STEP_TO_STEP -----------------------------
   "ChaosDB".Edge_Step1S := "ChaosDB".Step0 AND NOT "ChaosDB".Edge_Step1M;   // rising edge
   "ChaosDB".Edge_Step1M := "ChaosDB".Step0;
END_REGION

REGION Network 20
   RUNG wire#powerrail
      Contact( "ChaosDB".Edge_Step1S )
      wire#w1
      Coil( "ChaosDB".Step1 )
   END_RUNG
   RUNG wire#powerrail
      Contact( "ChaosDB".Step1 )
      I_Contact( "ChaosDB".Step1_Step2 )
   END_RUNG wire#w1
   // the same network as SCL:
   "ChaosDB".Step1 := "ChaosDB".Edge_Step1S OR ("ChaosDB".Step1 AND NOT "ChaosDB".Step1_Step2);
END_REGION

REGION Network 21
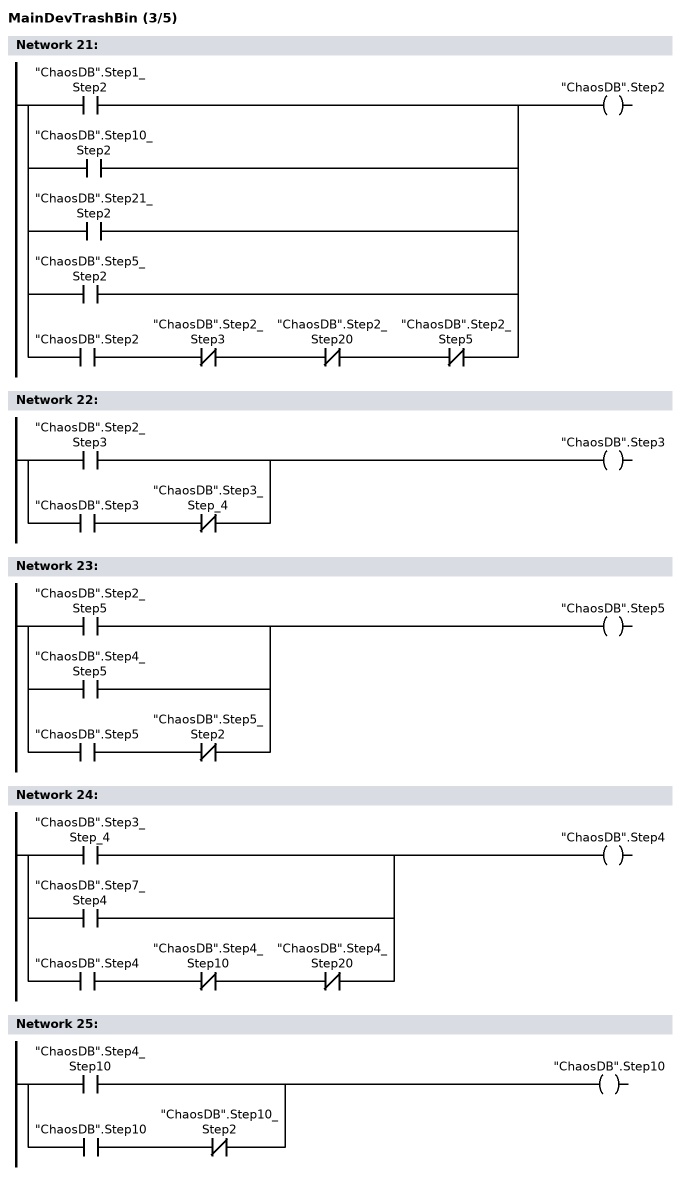
   RUNG wire#powerrail
      Contact( "ChaosDB".Step1_Step2 )
      wire#w1
      Coil( "ChaosDB".Step2 )
   END_RUNG
   RUNG wire#powerrail
      Contact( "ChaosDB".Step10_Step2 )
   END_RUNG wire#w1
   RUNG wire#powerrail
      Contact( "ChaosDB".Step21_Step2 )
   END_RUNG wire#w1
   RUNG wire#powerrail
      Contact( "ChaosDB".Step5_Step2 )
   END_RUNG wire#w1
   RUNG wire#powerrail
      Contact( "ChaosDB".Step2 )
      I_Contact( "ChaosDB".Step2_Step3 )
      I_Contact( "ChaosDB".Step2_Step20 )
      I_Contact( "ChaosDB".Step2_Step5 )
   END_RUNG wire#w1
   // the same network as SCL:
   "ChaosDB".Step2 := "ChaosDB".Step1_Step2 OR "ChaosDB".Step10_Step2 OR "ChaosDB".Step21_Step2 OR "ChaosDB".Step5_Step2 OR ("ChaosDB".Step2 AND NOT "ChaosDB".Step2_Step3 AND NOT "ChaosDB".Step2_Step20 AND NOT "ChaosDB".Step2_Step5);
END_REGION

REGION Network 22
   RUNG wire#powerrail
      Contact( "ChaosDB".Step2_Step3 )
      wire#w1
      Coil( "ChaosDB".Step3 )
   END_RUNG
   RUNG wire#powerrail
      Contact( "ChaosDB".Step3 )
      I_Contact( "ChaosDB".Step3_Step_4 )
   END_RUNG wire#w1
   // the same network as SCL:
   "ChaosDB".Step3 := "ChaosDB".Step2_Step3 OR ("ChaosDB".Step3 AND NOT "ChaosDB".Step3_Step_4);
END_REGION

REGION Network 23
   RUNG wire#powerrail
      Contact( "ChaosDB".Step2_Step5 )
      wire#w1
      Coil( "ChaosDB".Step5 )
   END_RUNG
   RUNG wire#powerrail
      Contact( "ChaosDB".Step4_Step5 )
   END_RUNG wire#w1
   RUNG wire#powerrail
      Contact( "ChaosDB".Step5 )
      I_Contact( "ChaosDB".Step5_Step2 )
   END_RUNG wire#w1
   // the same network as SCL:
   "ChaosDB".Step5 := "ChaosDB".Step2_Step5 OR "ChaosDB".Step4_Step5 OR ("ChaosDB".Step5 AND NOT "ChaosDB".Step5_Step2);
END_REGION

REGION Network 24
   RUNG wire#powerrail
      Contact( "ChaosDB".Step3_Step_4 )
      wire#w1
      Coil( "ChaosDB".Step4 )
   END_RUNG
   RUNG wire#powerrail
      Contact( "ChaosDB".Step7_Step4 )
   END_RUNG wire#w1
   RUNG wire#powerrail
      Contact( "ChaosDB".Step4 )
      I_Contact( "ChaosDB".Step4_Step10 )
      I_Contact( "ChaosDB".Step4_Step20 )
   END_RUNG wire#w1
   // the same network as SCL:
   "ChaosDB".Step4 := "ChaosDB".Step3_Step_4 OR "ChaosDB".Step7_Step4 OR ("ChaosDB".Step4 AND NOT "ChaosDB".Step4_Step10 AND NOT "ChaosDB".Step4_Step20);
END_REGION

REGION Network 25
   RUNG wire#powerrail
      Contact( "ChaosDB".Step4_Step10 )
      wire#w1
      Coil( "ChaosDB".Step10 )
   END_RUNG
   RUNG wire#powerrail
      Contact( "ChaosDB".Step10 )
      I_Contact( "ChaosDB".Step10_Step2 )
   END_RUNG wire#w1
   // the same network as SCL:
   "ChaosDB".Step10 := "ChaosDB".Step4_Step10 OR ("ChaosDB".Step10 AND NOT "ChaosDB".Step10_Step2);
END_REGION

REGION Network 26
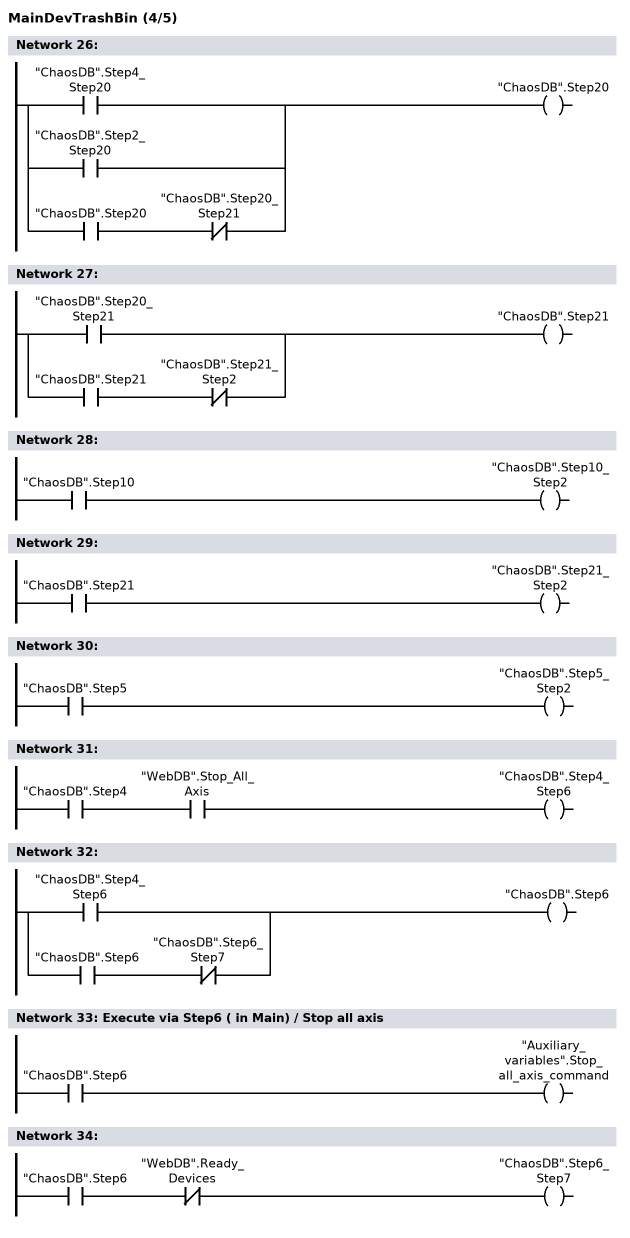
   RUNG wire#powerrail
      Contact( "ChaosDB".Step4_Step20 )
      wire#w1
      Coil( "ChaosDB".Step20 )
   END_RUNG
   RUNG wire#powerrail
      Contact( "ChaosDB".Step2_Step20 )
   END_RUNG wire#w1
   RUNG wire#powerrail
      Contact( "ChaosDB".Step20 )
      I_Contact( "ChaosDB".Step20_Step21 )
   END_RUNG wire#w1
   // the same network as SCL:
   "ChaosDB".Step20 := "ChaosDB".Step4_Step20 OR "ChaosDB".Step2_Step20 OR ("ChaosDB".Step20 AND NOT "ChaosDB".Step20_Step21);
END_REGION

REGION Network 27
   RUNG wire#powerrail
      Contact( "ChaosDB".Step20_Step21 )
      wire#w1
      Coil( "ChaosDB".Step21 )
   END_RUNG
   RUNG wire#powerrail
      Contact( "ChaosDB".Step21 )
      I_Contact( "ChaosDB".Step21_Step2 )
   END_RUNG wire#w1
   // the same network as SCL:
   "ChaosDB".Step21 := "ChaosDB".Step20_Step21 OR ("ChaosDB".Step21 AND NOT "ChaosDB".Step21_Step2);
END_REGION

REGION Network 28
   RUNG wire#powerrail
      Contact( "ChaosDB".Step10 )
      Coil( "ChaosDB".Step10_Step2 )
   END_RUNG
   // the same network as SCL:
   "ChaosDB".Step10_Step2 := "ChaosDB".Step10;
END_REGION

REGION Network 29
   RUNG wire#powerrail
      Contact( "ChaosDB".Step21 )
      Coil( "ChaosDB".Step21_Step2 )
   END_RUNG
   // the same network as SCL:
   "ChaosDB".Step21_Step2 := "ChaosDB".Step21;
END_REGION

REGION Network 30
   RUNG wire#powerrail
      Contact( "ChaosDB".Step5 )
      Coil( "ChaosDB".Step5_Step2 )
   END_RUNG
   // the same network as SCL:
   "ChaosDB".Step5_Step2 := "ChaosDB".Step5;
END_REGION

REGION Network 31
   RUNG wire#powerrail
      Contact( "ChaosDB".Step4 )
      Contact( "WebDB".Stop_All_Axis )
      Coil( "ChaosDB".Step4_Step6 )
   END_RUNG
   // the same network as SCL:
   "ChaosDB".Step4_Step6 := "ChaosDB".Step4 AND "WebDB".Stop_All_Axis;
END_REGION

REGION Network 32
   RUNG wire#powerrail
      Contact( "ChaosDB".Step4_Step6 )
      wire#w1
      Coil( "ChaosDB".Step6 )
   END_RUNG
   RUNG wire#powerrail
      Contact( "ChaosDB".Step6 )
      I_Contact( "ChaosDB".Step6_Step7 )
   END_RUNG wire#w1
   // the same network as SCL:
   "ChaosDB".Step6 := "ChaosDB".Step4_Step6 OR ("ChaosDB".Step6 AND NOT "ChaosDB".Step6_Step7);
END_REGION

REGION Network 33: Execute via Step6 ( in Main) / Stop all axis
   RUNG wire#powerrail
      Contact( "ChaosDB".Step6 )
      Coil( "Auxiliary_variables".Stop_all_axis_command )
   END_RUNG
   // the same network as SCL:
   "Auxiliary_variables".Stop_all_axis_command := "ChaosDB".Step6;
END_REGION

REGION Network 34
   RUNG wire#powerrail
      Contact( "ChaosDB".Step6 )
      I_Contact( "WebDB".Ready_Devices )
      Coil( "ChaosDB".Step6_Step7 )
   END_RUNG
   // the same network as SCL:
   "ChaosDB".Step6_Step7 := "ChaosDB".Step6 AND NOT "WebDB".Ready_Devices;
END_REGION

REGION Network 35
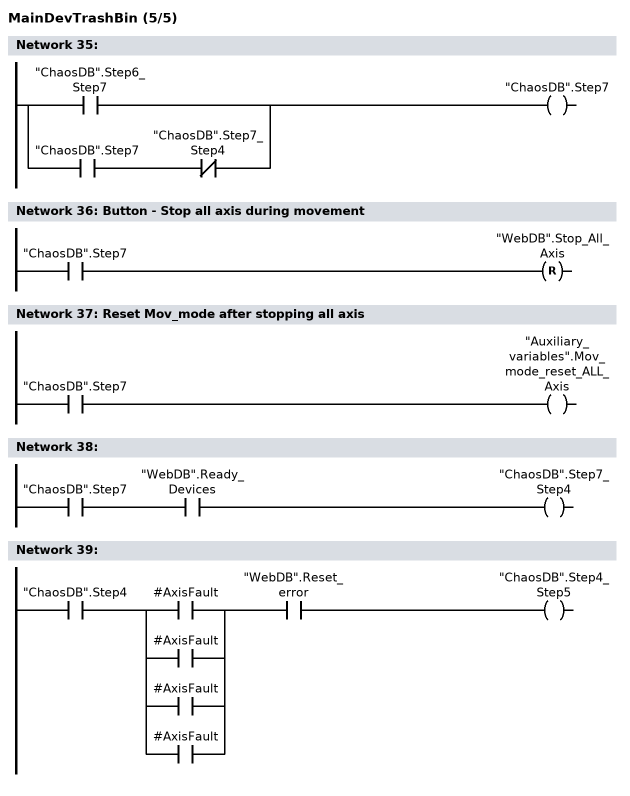
   RUNG wire#powerrail
      Contact( "ChaosDB".Step6_Step7 )
      wire#w1
      Coil( "ChaosDB".Step7 )
   END_RUNG
   RUNG wire#powerrail
      Contact( "ChaosDB".Step7 )
      I_Contact( "ChaosDB".Step7_Step4 )
   END_RUNG wire#w1
   // the same network as SCL:
   "ChaosDB".Step7 := "ChaosDB".Step6_Step7 OR ("ChaosDB".Step7 AND NOT "ChaosDB".Step7_Step4);
END_REGION

REGION Network 36: Button - Stop all axis during movement
   RUNG wire#powerrail
      Contact( "ChaosDB".Step7 )
      R_Coil( "WebDB".Stop_All_Axis )
   END_RUNG
   // the same network as SCL:
   IF "ChaosDB".Step7 THEN "WebDB".Stop_All_Axis := FALSE; END_IF;
END_REGION

REGION Network 37: Reset Mov_mode after stopping all axis
   RUNG wire#powerrail
      Contact( "ChaosDB".Step7 )
      Coil( "Auxiliary_variables".Mov_mode_reset_ALL_Axis )
   END_RUNG
   // the same network as SCL:
   "Auxiliary_variables".Mov_mode_reset_ALL_Axis := "ChaosDB".Step7;
END_REGION

REGION Network 38
   RUNG wire#powerrail
      Contact( "ChaosDB".Step7 )
      Contact( "WebDB".Ready_Devices )
      Coil( "ChaosDB".Step7_Step4 )
   END_RUNG
   // the same network as SCL:
   "ChaosDB".Step7_Step4 := "ChaosDB".Step7 AND "WebDB".Ready_Devices;
END_REGION

REGION Network 39
   RUNG wire#powerrail
      Contact( "ChaosDB".Step4 )
      wire#w1
      Contact( #AxisFault )
      wire#w2
      Contact( "WebDB".Reset_error )
      Coil( "ChaosDB".Step4_Step5 )
   END_RUNG
   RUNG wire#w1
      Contact( #AxisFault )
   END_RUNG wire#w2
   RUNG wire#w1
      Contact( #AxisFault )
   END_RUNG wire#w2
   RUNG wire#w1
      Contact( #AxisFault )
   END_RUNG wire#w2
   // the same network as SCL:
   "ChaosDB".Step4_Step5 := "ChaosDB".Step4 AND (#AxisFault OR #AxisFault OR #AxisFault OR #AxisFault) AND "WebDB".Reset_error;
END_REGION
END_FUNCTION

FUNCTION "Enable-Axis" : Void   // FC3, LAD
{ S7_Optimized_Access := 'TRUE' }
AUTHOR : HenriP
VERSION : 0.1
   VAR_INPUT
      Enable : Bool;
      "E-STOP" : Bool;
      Stop : Bool;
      Halt : Bool;
   END_VAR
   VAR_OUTPUT
      FestoStop : Bool;
      FestoEnable : Bool;
      FestoHalt : Bool;
   END_VAR
BEGIN

REGION Network 1: Festo Enable
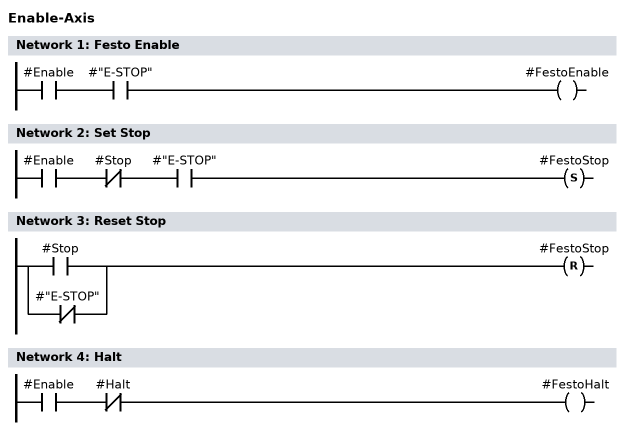
   RUNG wire#powerrail
      Contact( #Enable )
      Contact( #"E-STOP" )
      Coil( #FestoEnable )
   END_RUNG
   // the same network as SCL:
   #FestoEnable := #Enable AND #"E-STOP";
END_REGION

REGION Network 2: Set Stop
   RUNG wire#powerrail
      Contact( #Enable )
      I_Contact( #Stop )
      Contact( #"E-STOP" )
      S_Coil( #FestoStop )
   END_RUNG
   // the same network as SCL:
   IF #Enable AND NOT #Stop AND #"E-STOP" THEN #FestoStop := TRUE; END_IF;
END_REGION

REGION Network 3: Reset Stop
   RUNG wire#powerrail
      Contact( #Stop )
      wire#w1
      R_Coil( #FestoStop )
   END_RUNG
   RUNG wire#powerrail
      I_Contact( #"E-STOP" )
   END_RUNG wire#w1
   // the same network as SCL:
   IF #Stop OR NOT #"E-STOP" THEN #FestoStop := FALSE; END_IF;
END_REGION

REGION Network 4: Halt
   RUNG wire#powerrail
      Contact( #Enable )
      I_Contact( #Halt )
      Coil( #FestoHalt )
   END_RUNG
   // the same network as SCL:
   #FestoHalt := #Enable AND NOT #Halt;
END_REGION
END_FUNCTION

FUNCTION "LED" : Void   // FC6, LAD
{ S7_Optimized_Access := 'TRUE' }
AUTHOR : HenriP
VERSION : 0.1
   VAR_INPUT
      Green : Bool;
      GreenBlink : Bool;
      Red : Bool;
      RedBlink : Bool;
      RedGreen : Bool;
   END_VAR
   VAR_OUTPUT
      "Led Green" : Bool;
      "Led Red" : Bool;
   END_VAR
   VAR_TEMP
      RedGreenBlinkTemp : Bool;
      RedBlinkTemp : Bool;
      GreenBlinkTemp : Bool;
   END_VAR
BEGIN

REGION Network 1: Green Led
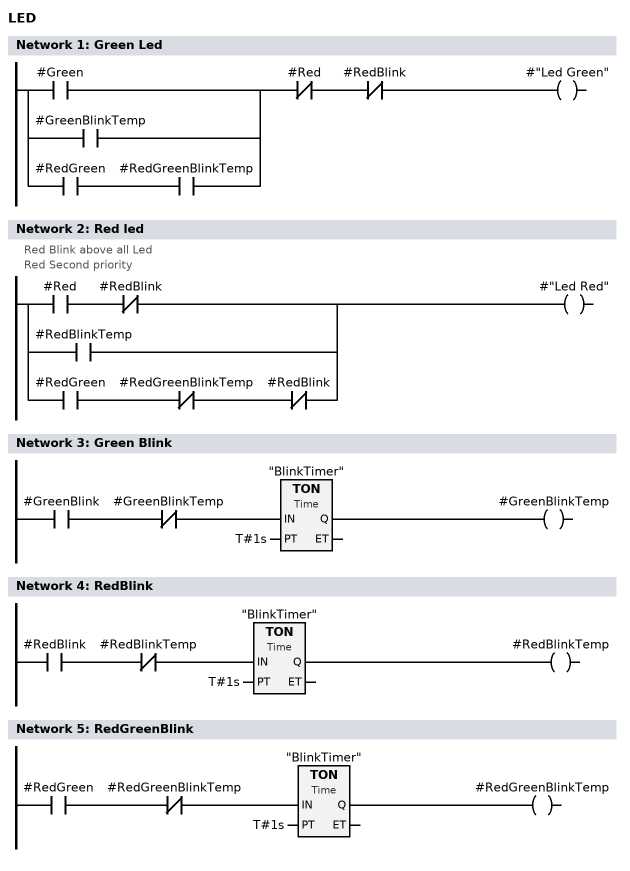
   RUNG wire#powerrail
      Contact( #Green )
      wire#w1
      I_Contact( #Red )
      I_Contact( #RedBlink )
      Coil( #"Led Green" )
   END_RUNG
   RUNG wire#powerrail
      Contact( #GreenBlinkTemp )
   END_RUNG wire#w1
   RUNG wire#powerrail
      Contact( #RedGreen )
      Contact( #RedGreenBlinkTemp )
   END_RUNG wire#w1
   // the same network as SCL:
   #"Led Green" := (#Green OR #GreenBlinkTemp OR (#RedGreen AND #RedGreenBlinkTemp)) AND NOT #Red AND NOT #RedBlink;
END_REGION

REGION Network 2: Red led
   // Red Blink above all Led
   // Red Second priority
   RUNG wire#powerrail
      Contact( #Red )
      I_Contact( #RedBlink )
      wire#w1
      Coil( #"Led Red" )
   END_RUNG
   RUNG wire#powerrail
      Contact( #RedBlinkTemp )
   END_RUNG wire#w1
   RUNG wire#powerrail
      Contact( #RedGreen )
      I_Contact( #RedGreenBlinkTemp )
      I_Contact( #RedBlink )
   END_RUNG wire#w1
   // the same network as SCL:
   #"Led Red" := (#Red AND NOT #RedBlink) OR #RedBlinkTemp OR (#RedGreen AND NOT #RedGreenBlinkTemp AND NOT #RedBlink);
END_REGION

REGION Network 3: Green Blink
   RUNG wire#powerrail
      Contact( #GreenBlink )
      I_Contact( #GreenBlinkTemp )
      { S7_Templates := "time_type := Time" } "BlinkTimer".TON(pt := T#1s, et =>)
      Coil( #GreenBlinkTemp )
   END_RUNG
   // the same network as SCL:
   "BlinkTimer".TON(IN := #GreenBlink AND NOT #GreenBlinkTemp, PT := T#1s);
   #GreenBlinkTemp := "BlinkTimer".Q;
END_REGION

REGION Network 4: RedBlink
   RUNG wire#powerrail
      Contact( #RedBlink )
      I_Contact( #RedBlinkTemp )
      { S7_Templates := "time_type := Time" } "BlinkTimer".TON(pt := T#1s, et =>)
      Coil( #RedBlinkTemp )
   END_RUNG
   // the same network as SCL:
   "BlinkTimer".TON(IN := #RedBlink AND NOT #RedBlinkTemp, PT := T#1s);
   #RedBlinkTemp := "BlinkTimer".Q;
END_REGION

REGION Network 5: RedGreenBlink
   RUNG wire#powerrail
      Contact( #RedGreen )
      I_Contact( #RedGreenBlinkTemp )
      { S7_Templates := "time_type := Time" } "BlinkTimer".TON(pt := T#1s, et =>)
      Coil( #RedGreenBlinkTemp )
   END_RUNG
   // the same network as SCL:
   "BlinkTimer".TON(IN := #RedGreen AND NOT #RedGreenBlinkTemp, PT := T#1s);
   #RedGreenBlinkTemp := "BlinkTimer".Q;
END_REGION
END_FUNCTION

FUNCTION "RollerV2" : Void   // FC16, LAD
{ S7_Optimized_Access := 'TRUE' }
AUTHOR : HenriP
VERSION : 0.1
// Module behave as a flip flip switch for the Start and Stop Command
   VAR_INPUT
      SystemON : Bool;
   END_VAR
   VAR_IN_OUT
      Start : Bool;
      Stop : Bool;
      ORoller : Bool;
   END_VAR
BEGIN

REGION Network 1: RollerON
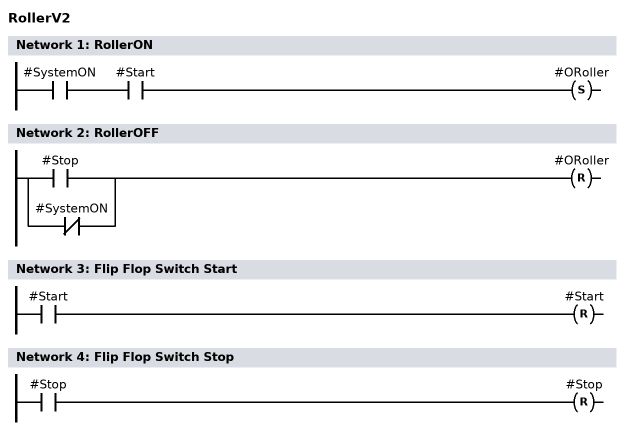
   RUNG wire#powerrail
      Contact( #SystemON )
      Contact( #Start )
      S_Coil( #ORoller )
   END_RUNG
   // the same network as SCL:
   IF #SystemON AND #Start THEN #ORoller := TRUE; END_IF;
END_REGION

REGION Network 2: RollerOFF
   RUNG wire#powerrail
      Contact( #Stop )
      wire#w1
      R_Coil( #ORoller )
   END_RUNG
   RUNG wire#powerrail
      I_Contact( #SystemON )
   END_RUNG wire#w1
   // the same network as SCL:
   IF #Stop OR NOT #SystemON THEN #ORoller := FALSE; END_IF;
END_REGION

REGION Network 3: Flip Flop Switch Start
   RUNG wire#powerrail
      Contact( #Start )
      R_Coil( #Start )
   END_RUNG
   // the same network as SCL:
   IF #Start THEN #Start := FALSE; END_IF;
END_REGION

REGION Network 4: Flip Flop Switch Stop
   RUNG wire#powerrail
      Contact( #Stop )
      R_Coil( #Stop )
   END_RUNG
   // the same network as SCL:
   IF #Stop THEN #Stop := FALSE; END_IF;
END_REGION
END_FUNCTION

FUNCTION "MotionController" : Void   // FC14, LAD
{ S7_Optimized_Access := 'TRUE' }
AUTHOR : HenriP
VERSION : 0.1
   VAR_INPUT
      "E-STOP" : Bool;
      JogPBtn : Bool;
      JogNBtn : Bool;
      TargetRange : DInt;
      PosMax : DInt;
      PosMin : DInt;
      AxisColision : Bool;
      DoorSensor : Bool;
   END_VAR
   VAR_OUTPUT
      AxisOutput : Struct
         DriveEnabled : Bool;
         Ready : Bool;
         Warning : Bool;
         Fault : Bool;
         SupplyVoltPresent : Bool;
         ControlFCT_HMI : Bool;
         StateOPM : Int;
         HaltNotActive : Bool;
         AckStart : Bool;
         MC : Bool;
         AckTeach : Bool;
         DriveMoving : Bool;
         DragError : Bool;
         StandStillControl : Bool;
         HomingValid : Bool;
         ActualRecordNo : Int;
         RC1 : Bool;
         RCC : Bool;
         VelocityLimitReached : Bool;
         StrokeLimitReached : Bool;
         FunctionIsActive : Bool;
         ActualFunctionNumber : Int;
         ActualFunctionGroup : Int;
         ActualPosition : DInt;
         ActualVelocity : DInt;
         ActualForce : DInt;
         ActualRotRamp : DInt;
         ActualRotSpeed : DInt;
      END_STRUCT;
      TargetReached : Bool;
      Overange : Bool;
   END_VAR
   VAR_IN_OUT
      AxisInput : Struct
         EnableDrive : Bool;
         Stop : Bool;
         Halt : Bool;
         Brake : Bool;
         ResetFault : Bool;
         HMIAccessLocked : Bool;
         OPM : Int;
         StartTask : Bool;
         StartHoming : Bool;
         JogPos : Bool;
         JogNeg : Bool;
         TeachActValue : Bool;
         ClearRemPos : Bool;
         Relative : Bool;
         DeactivateStrokeLimit : Bool;
         ExecuteFunction : Bool;
         RecordNo : Int;
         SetFunctionNumber : Int;
         SetFunctionGroup : Int;
         SetValueVelocity : DInt;
         SetValuePosition : DInt;
         SetValueForceRamp : DInt;
         SetValueForce : DInt;
         SetValueRotRamp : DInt;
         SetValueRotSpeed : DInt;
      END_STRUCT;
      FestoDB : "FHPP_CTRL";
      TaskE : Bool;
      TaskM : Bool;
   END_VAR
   VAR_TEMP
      TargetDistance : DInt;
      ErrorValue : Int;
      Pos : DInt;
      PosAdd : DInt;
      PosSub : DInt;
      TaskEBis : Bool;
      JogPOv : DInt;
   END_VAR
   VAR_TEMP   // added for the SCL form of the ladder/FBD networks
      _w1 : Bool;
      _w2 : Bool;
   END_VAR
BEGIN

REGION Network 1: Enable Axis - Stop Control
   // For safety reason the Safety torque control is on a special loop , Emergency stop may move there too
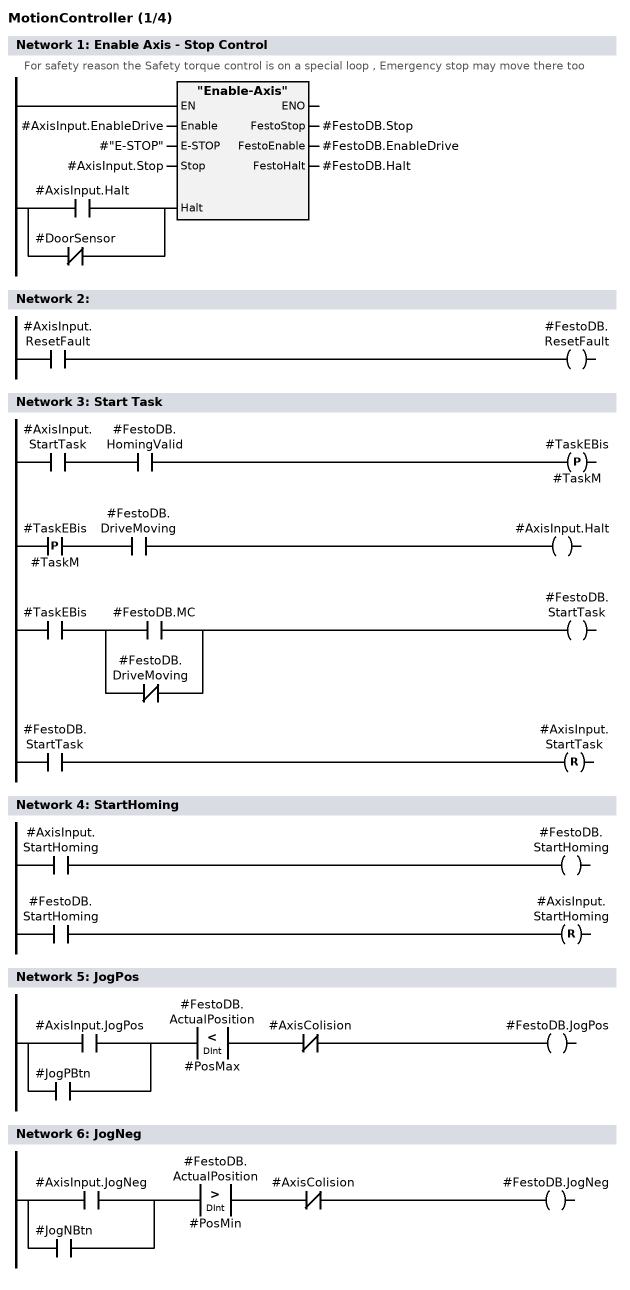
   RUNG wire#powerrail
      "Enable-Axis"(Halt := wire#w1, Enable := #AxisInput.EnableDrive, "E-STOP" := #"E-STOP", Stop := #AxisInput.Stop, FestoStop => #FestoDB.Stop, FestoEnable => #FestoDB.EnableDrive, FestoHalt => #FestoDB.Halt)
   END_RUNG
   RUNG wire#powerrail
      Contact( #AxisInput.Halt )
   END_RUNG wire#w1
   RUNG wire#powerrail
      I_Contact( #DoorSensor )
   END_RUNG wire#w1
   // the same network as SCL:
   "Enable-Axis"(Enable := #AxisInput.EnableDrive,
                 "E-STOP" := #"E-STOP",
                 Stop := #AxisInput.Stop,
                 Halt := #AxisInput.Halt OR NOT #DoorSensor,
                 FestoStop => #FestoDB.Stop,
                 FestoEnable => #FestoDB.EnableDrive,
                 FestoHalt => #FestoDB.Halt);
END_REGION

REGION Network 2
   RUNG wire#powerrail
      Contact( #AxisInput.ResetFault )
      Coil( #FestoDB.ResetFault )
   END_RUNG
   // the same network as SCL:
   #FestoDB.ResetFault := #AxisInput.ResetFault;
END_REGION

REGION Network 3: Start Task
   #_w1 := #AxisInput.StartTask AND #FestoDB.HomingValid;
   #TaskEBis := #_w1 AND NOT #TaskM;   // rising edge
   #TaskM := #_w1;
   #_w2 := #TaskEBis AND NOT #TaskM;   // rising edge of #TaskEBis
   #TaskM := #TaskEBis;
   #AxisInput.Halt := #_w2 AND #FestoDB.DriveMoving;
   #FestoDB.StartTask := #TaskEBis AND (#FestoDB.MC OR NOT #FestoDB.DriveMoving);
   IF #FestoDB.StartTask THEN #AxisInput.StartTask := FALSE; END_IF;
END_REGION

REGION Network 4: StartHoming
   RUNG wire#powerrail
      Contact( #AxisInput.StartHoming )
      Coil( #FestoDB.StartHoming )
   END_RUNG
   RUNG wire#powerrail
      Contact( #FestoDB.StartHoming )
      R_Coil( #AxisInput.StartHoming )
   END_RUNG
   // the same network as SCL:
   #FestoDB.StartHoming := #AxisInput.StartHoming;
   IF #FestoDB.StartHoming THEN #AxisInput.StartHoming := FALSE; END_IF;
END_REGION

REGION Network 5: JogPos
   RUNG wire#powerrail
      Contact( #AxisInput.JogPos )
      wire#w1
      { S7_Templates := "SrcType := DInt" } LT_Contact(in1 := #FestoDB.ActualPosition, in2 := #PosMax)
      I_Contact( #AxisColision )
      Coil( #FestoDB.JogPos )
   END_RUNG
   RUNG wire#powerrail
      Contact( #JogPBtn )
   END_RUNG wire#w1
   // the same network as SCL:
   #FestoDB.JogPos := (#AxisInput.JogPos OR #JogPBtn) AND (#FestoDB.ActualPosition < #PosMax) AND NOT #AxisColision;
END_REGION

REGION Network 6: JogNeg
   RUNG wire#powerrail
      Contact( #AxisInput.JogNeg )
      wire#w1
      { S7_Templates := "SrcType := DInt" } GT_Contact(in1 := #FestoDB.ActualPosition, in2 := #PosMin)
      I_Contact( #AxisColision )
      Coil( #FestoDB.JogNeg )
   END_RUNG
   RUNG wire#powerrail
      Contact( #JogNBtn )
   END_RUNG wire#w1
   // the same network as SCL:
   #FestoDB.JogNeg := (#AxisInput.JogNeg OR #JogNBtn) AND (#FestoDB.ActualPosition > #PosMin) AND NOT #AxisColision;
END_REGION

REGION Network 7: Relative Input Command
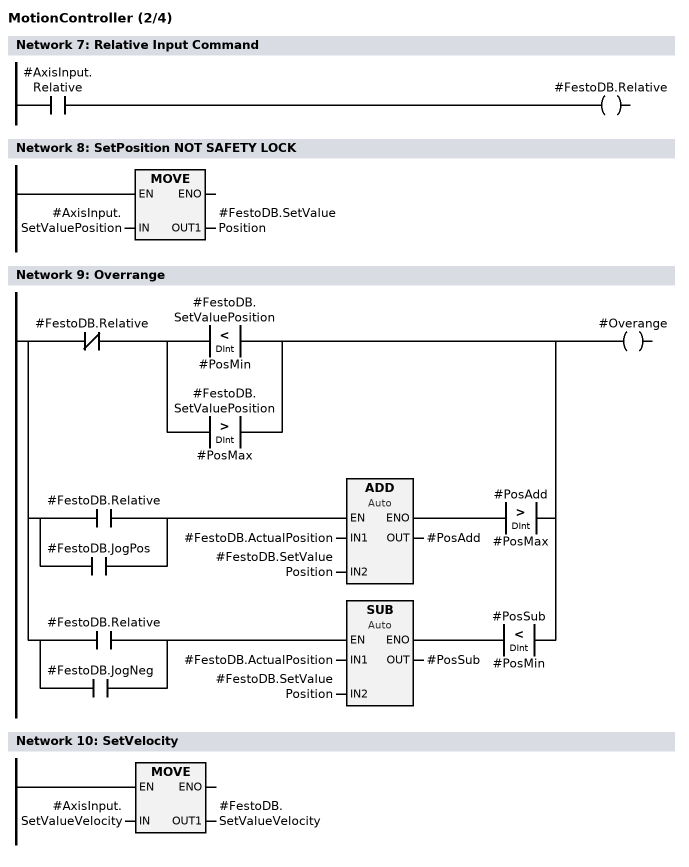
   RUNG wire#powerrail
      Contact( #AxisInput.Relative )
      Coil( #FestoDB.Relative )
   END_RUNG
   // the same network as SCL:
   #FestoDB.Relative := #AxisInput.Relative;
END_REGION

REGION Network 8: SetPosition NOT SAFETY LOCK
   RUNG wire#powerrail
      Move(in := #AxisInput.SetValuePosition, out1 => #FestoDB.SetValuePosition)
   END_RUNG
   // the same network as SCL:
   #FestoDB.SetValuePosition := #AxisInput.SetValuePosition;
END_REGION

REGION Network 9: Overrange
   RUNG wire#powerrail
      I_Contact( #FestoDB.Relative )
      wire#w1
      { S7_Templates := "SrcType := DInt" } LT_Contact(in1 := #FestoDB.SetValuePosition, in2 := #PosMin)
      wire#w2
      Coil( #Overange )
   END_RUNG
   RUNG wire#w1
      { S7_Templates := "SrcType := DInt" } GT_Contact(in1 := #FestoDB.SetValuePosition, in2 := #PosMax)
   END_RUNG wire#w2
   RUNG wire#powerrail
      Contact( #FestoDB.Relative )
      wire#w3
      Add(in1 := #FestoDB.ActualPosition, in2 := #FestoDB.SetValuePosition, out => #PosAdd)
      { S7_Templates := "SrcType := DInt" } GT_Contact(in1 := #PosAdd, in2 := #PosMax)
   END_RUNG wire#w2
   RUNG wire#powerrail
      Contact( #FestoDB.JogPos )
   END_RUNG wire#w3
   RUNG wire#powerrail
      Contact( #FestoDB.Relative )
      wire#w4
      Sub(in1 := #FestoDB.ActualPosition, in2 := #FestoDB.SetValuePosition, out => #PosSub)
      { S7_Templates := "SrcType := DInt" } LT_Contact(in1 := #PosSub, in2 := #PosMin)
   END_RUNG wire#w2
   RUNG wire#powerrail
      Contact( #FestoDB.JogNeg )
   END_RUNG wire#w4
   // the same network as SCL:
   #_w1 := #FestoDB.Relative OR #FestoDB.JogPos;
   IF #_w1 THEN #PosAdd := #FestoDB.ActualPosition + #FestoDB.SetValuePosition; END_IF;
   #_w2 := #FestoDB.Relative OR #FestoDB.JogNeg;
   IF #_w2 THEN #PosSub := #FestoDB.ActualPosition - #FestoDB.SetValuePosition; END_IF;
   #Overange := (NOT #FestoDB.Relative AND ((#FestoDB.SetValuePosition < #PosMin) OR (#FestoDB.SetValuePosition > #PosMax))) OR (#_w1 AND (#PosAdd > #PosMax)) OR (#_w2 AND (#PosSub < #PosMin));
END_REGION

REGION Network 10: SetVelocity
   RUNG wire#powerrail
      Move(in := #AxisInput.SetValueVelocity, out1 => #FestoDB.SetValueVelocity)
   END_RUNG
   // the same network as SCL:
   #FestoDB.SetValueVelocity := #AxisInput.SetValueVelocity;
END_REGION

